KUKA KRL program: PPR-bot-01.src

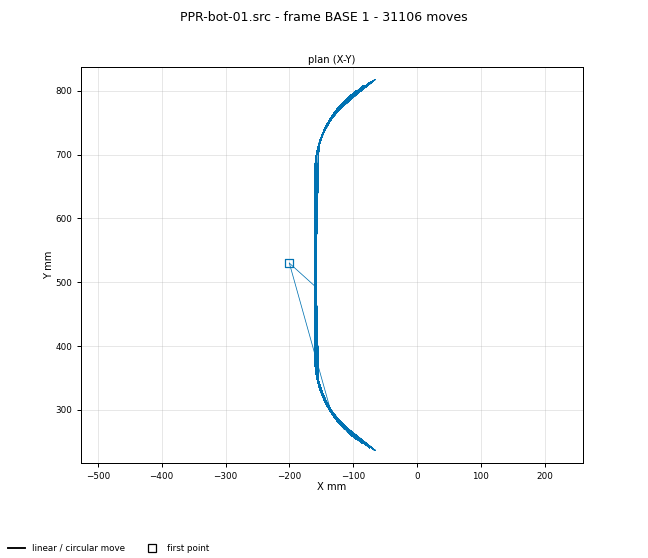
[picture p0: tool path of PPR-bot-01.src in frame BASE 1, 31106 of 31107 moves have a stored position in this frame; points joined in program order, loops and branches not executed]
&ACCESS RVEO
&REL 11
&PARAM TEMPLATE = C:\KRC\Roboter\Template\vorgabe
&PARAM EDITMASK = *
DEF variable_helical2( )
;FOLD INI
  ;FOLD BASISTECH INI
    GLOBAL INTERRUPT DECL 3 WHEN $STOPMESS==TRUE DO IR_STOPM ( )
    INTERRUPT ON 3
    BAS (#INITMOV,0 )
  ;ENDFOLD (BASISTECH INI)
 ;FOLD USER INI


    ;Make your modifications here
  ;ENDFOLD (USER INI)
;ENDFOLD (INI)
ACTION(#AXIS_RESET,34,1000,#NOERROR,ERROR_CODE)
;FOLD PTP HOME  Vel= 100 % DEFAULT;%{PE}%MKUKATPBASIS,%CMOVE,%VPTP,%P 1:PTP, 2:HOME, 3:, 5:100, 7:DEFAULT
$BWDSTART = FALSE
PDAT_ACT=PDEFAULT
FDAT_ACT=FHOME
BAS (#PTP_PARAMS,100 )
$H_POS=XHOME
PTP  XHOME
;ENDFOLD
BAS(#TOOL,1)
BAS(#BASE,1)
$VEL_AXIS[1]=100
$VEL_AXIS[2]=100
$VEL_AXIS[3]=100
$VEL_AXIS[4]=100
$VEL_AXIS[5]=100
$VEL_AXIS[6]=100
$VEL_EXTAX[1]=100
$VEL_EXTAX[2]=100

$ACC_AXIS[1]=100
$ACC_AXIS[2]=100
$ACC_AXIS[3]=100
$ACC_AXIS[4]=100
$ACC_AXIS[5]=100
$ACC_AXIS[6]=100
$ACC_EXTAX[1]=100
$ACC_EXTAX[2]=100

;;;;;;;;; postprocessing parameters (date 2024-01-25T18:13:03.555540)
; qxconst: -159.99
; qxconstarcys: -147.5,141.5
; qE3offset: 0.00
; qyoffset: 530.00
; qswitchsplit: 3
; qthinningtol: 0.2010
;;;;;;;;;

SLIN {X  -200.000, Y  +530.000, Z    +0.000, A    +0.000, E1    +0.000, E3    +0.000, E4    +0.000}

SLIN {X  -134.349, Y  +295.626, Z    +0.000, E1   +74.322, E3  -296.855}
HALT
SPLINE
SPL {X  -131.287, Y  +291.064, Z    +0.000, E1   +73.972, E3  -292.043}
SPL {X  -128.265, Y  +286.871, Z    +0.000, E1   +73.613, E3  -287.587}
SPL {X  -125.161, Y  +282.843, Z    +0.000, E1   +73.232, E3  -283.315}
SPL {X  -122.038, Y  +279.042, Z    +0.000, E1   +72.832, E3  -279.335}
SPL {X  -118.642, Y  +275.165, Z    +0.000, E1   +72.381, E3  -275.372}
SPL {X   -66.040, Y  +236.776, Z    +0.000, E1   +55.694, E3  -114.008}
ENDSPLINE

SPLINE
SPL {X  -127.452, Y  +285.790, Z    +0.000, E1   +56.591, E3   +59.937}
SPL {X  -151.591, Y  +331.344, Z    +0.000, E1   +43.870, E3   +76.036}
SPL {X  -158.135, Y  +358.205, Z    +0.000, E1   +26.984, E3   +79.764}
SPL {X  -159.602, Y  +371.361, Z    +0.000, E1   +14.835, E3   +80.660}
SPL {X  -159.981, Y  +380.818, Z    +0.000, E1    +4.512, E3   +80.938}
SPL {X  -159.990, Y  +384.681, Z    +0.000, E1    -0.222, E3   +80.967}
SPL {X  -159.990, Y  +387.626, Z    +0.000, E1    -8.190, E3   +80.995}
SPL {X  -159.990, Y  +390.340, Z    +0.000, E1   -15.987, E3   +81.060}
SPL {X  -159.990, Y  +394.216, Z    +0.000, E1   -27.062, E3   +81.222}
SPL {X  -159.990, Y  +399.855, Z    +0.000, E1   -40.916, E3   +81.593}
SPL {X  -159.990, Y  +405.475, Z    +0.000, E1   -51.039, E3   +82.110}
SPL {X  -159.990, Y  +414.231, Z    +0.000, E1   -60.575, E3   +83.294}
SPL {X  -159.990, Y  +462.953, Z    +0.000, E1   -73.611, E3   +95.033}
SPL {X  -153.839, Y  +715.436, Z    +0.000, E1   -75.884, E3  +197.463}
SPL {X  -148.840, Y  +730.182, Z    +0.000, E1   -75.434, E3  +210.040}
SPL {X  -143.409, Y  +742.426, Z    +0.000, E1   -74.905, E3  +221.552}
SPL {X  -139.557, Y  +749.735, Z    +0.000, E1   -74.483, E3  +228.900}
SPL {X  -136.371, Y  +755.165, Z    +0.000, E1   -74.152, E3  +234.446}
SPL {X  -133.102, Y  +760.274, Z    +0.000, E1   -73.777, E3  +239.831}
SPL {X  -128.975, Y  +766.169, Z    +0.000, E1   -73.313, E3  +246.106}
SPL {X  -124.947, Y  +771.425, Z    +0.000, E1   -72.782, E3  +251.799}
SPL {X  -121.698, Y  +775.357, Z    +0.000, E1   -72.353, E3  +255.994}
SPL {X  -118.622, Y  +778.858, Z    +0.000, E1   -71.924, E3  +259.620}
SPL {X   -66.171, Y  +817.165, Z    +0.000, E1   -56.016, E3  +410.978}
ENDSPLINE

SPLINE
SPL {X  -126.418, Y  +769.557, Z    +0.000, E1   -57.118, E3  +594.219}
SPL {X  -145.244, Y  +738.589, Z    +0.000, E1   -50.405, E3  +607.461}
SPL {X  -150.151, Y  +726.741, Z    +0.000, E1   -46.068, E3  +610.388}
SPL {X  -156.642, Y  +704.059, Z    +0.000, E1   -33.659, E3  +614.017}
SPL {X  -159.317, Y  +686.157, Z    +0.000, E1   -18.660, E3  +615.507}
SPL {X  -159.907, Y  +676.666, Z    +0.000, E1    -8.555, E3  +615.905}
SPL {X  -159.990, Y  +669.586, Z    +0.000, E1    -0.216, E3  +615.996}
SPL {X  -159.990, Y  +667.794, Z    +0.000, E1    +4.255, E3  +616.007}
SPL {X  -159.990, Y  +664.091, Z    +0.000, E1   +14.928, E3  +616.079}
SPL {X  -159.990, Y  +658.301, Z    +0.000, E1   +31.283, E3  +616.332}
SPL {X  -159.990, Y  +650.845, Z    +0.000, E1   +47.892, E3  +616.877}
SPL {X  -159.990, Y  +640.730, Z    +0.000, E1   +60.297, E3  +618.078}
SPL {X  -159.990, Y  +620.478, Z    +0.000, E1   +70.026, E3  +621.891}
SPL {X  -159.990, Y  +573.021, Z    +0.000, E1   +74.619, E3  +635.835}
SPL {X  -155.476, Y  +344.766, Z    +0.000, E1   +76.025, E3  +727.806}
SPL {X  -153.405, Y  +337.073, Z    +0.000, E1   +75.847, E3  +733.861}
SPL {X  -150.223, Y  +327.456, Z    +0.000, E1   +75.573, E3  +741.947}
SPL {X  -136.549, Y  +299.126, Z    +0.000, E1   +77.537, E3  +734.837}
ENDSPLINE

SPLINE
SPL {X  -136.626, Y  +299.252, Z    +0.000, E1   +76.314, E3  +746.487}
ENDSPLINE

SPLINE
SPL {X  -135.890, Y  +298.057, Z    +0.000, E1   +75.040, E3  +757.836}
SPL {X  -134.349, Y  +295.626, Z    +0.000, E1   +74.322, E3  +764.683}
SPL {X  -131.287, Y  +291.064, Z    +0.000, E1   +73.972, E3  +769.496}
SPL {X  -128.265, Y  +286.871, Z    +0.000, E1   +73.613, E3  +773.952}
SPL {X  -125.161, Y  +282.843, Z    +0.000, E1   +73.232, E3  +778.224}
SPL {X  -122.038, Y  +279.042, Z    +0.000, E1   +72.832, E3  +782.204}
SPL {X  -118.642, Y  +275.165, Z    +0.000, E1   +72.381, E3  +786.167}
SPL {X   -66.040, Y  +236.776, Z    +0.000, E1   +55.694, E3  +947.530}
ENDSPLINE

SPLINE
SPL {X  -127.452, Y  +285.790, Z    +0.000, E1   +56.591, E3 +1121.476}
SPL {X  -148.001, Y  +321.733, Z    +0.000, E1   +47.810, E3 +1135.579}
SPL {X  -154.604, Y  +341.337, Z    +0.000, E1   +38.630, E3 +1139.353}
SPL {X  -158.135, Y  +358.205, Z    +0.000, E1   +26.984, E3 +1141.302}
SPL {X  -159.602, Y  +371.361, Z    +0.000, E1   +14.835, E3 +1142.198}
SPL {X  -159.981, Y  +380.818, Z    +0.000, E1    +4.512, E3 +1142.476}
SPL {X  -159.990, Y  +384.681, Z    +0.000, E1    -0.222, E3 +1142.505}
SPL {X  -159.990, Y  +387.626, Z    +0.000, E1    -8.190, E3 +1142.534}
SPL {X  -159.990, Y  +390.340, Z    +0.000, E1   -15.987, E3 +1142.598}
SPL {X  -159.990, Y  +394.216, Z    +0.000, E1   -27.062, E3 +1142.760}
SPL {X  -159.990, Y  +399.855, Z    +0.000, E1   -40.916, E3 +1143.131}
SPL {X  -159.990, Y  +405.475, Z    +0.000, E1   -51.039, E3 +1143.648}
SPL {X  -159.990, Y  +414.231, Z    +0.000, E1   -60.575, E3 +1144.832}
SPL {X  -159.990, Y  +462.953, Z    +0.000, E1   -73.611, E3 +1156.571}
SPL {X  -153.839, Y  +715.436, Z    +0.000, E1   -75.884, E3 +1259.002}
SPL {X  -149.923, Y  +727.355, Z    +0.000, E1   -75.515, E3 +1269.112}
SPL {X  -145.995, Y  +736.939, Z    +0.000, E1   -75.150, E3 +1277.846}
SPL {X  -141.012, Y  +747.080, Z    +0.000, E1   -74.661, E3 +1287.699}
SPL {X  -136.371, Y  +755.165, Z    +0.000, E1   -74.152, E3 +1295.984}
SPL {X  -133.102, Y  +760.274, Z    +0.000, E1   -73.777, E3 +1301.369}
SPL {X  -128.975, Y  +766.169, Z    +0.000, E1   -73.313, E3 +1307.645}
SPL {X  -124.947, Y  +771.425, Z    +0.000, E1   -72.782, E3 +1313.338}
SPL {X  -121.698, Y  +775.357, Z    +0.000, E1   -72.353, E3 +1317.532}
SPL {X  -118.622, Y  +778.858, Z    +0.000, E1   -71.924, E3 +1321.158}
SPL {X   -66.171, Y  +817.165, Z    +0.000, E1   -56.016, E3 +1472.517}
ENDSPLINE

SPLINE
SPL {X  -126.418, Y  +769.557, Z    +0.000, E1   -57.118, E3 +1655.758}
SPL {X  -145.244, Y  +738.589, Z    +0.000, E1   -50.405, E3 +1668.999}
SPL {X  -150.151, Y  +726.741, Z    +0.000, E1   -46.068, E3 +1671.926}
SPL {X  -156.642, Y  +704.059, Z    +0.000, E1   -33.659, E3 +1675.555}
SPL {X  -159.317, Y  +686.157, Z    +0.000, E1   -18.660, E3 +1677.046}
SPL {X  -159.973, Y  +673.799, Z    +0.000, E1    -5.345, E3 +1677.494}
SPL {X  -159.990, Y  +669.500, Z    +0.000, E1    +0.000, E3 +1677.534}
SPL {X  -159.990, Y  +667.794, Z    +0.000, E1    +4.255, E3 +1677.546}
SPL {X  -159.990, Y  +664.091, Z    +0.000, E1   +14.928, E3 +1677.618}
SPL {X  -159.990, Y  +658.301, Z    +0.000, E1   +31.283, E3 +1677.870}
SPL {X  -159.990, Y  +650.845, Z    +0.000, E1   +47.892, E3 +1678.415}
SPL {X  -159.990, Y  +640.730, Z    +0.000, E1   +60.297, E3 +1679.617}
SPL {X  -159.990, Y  +620.478, Z    +0.000, E1   +70.026, E3 +1683.430}
SPL {X  -159.990, Y  +573.021, Z    +0.000, E1   +74.619, E3 +1697.374}
SPL {X  -154.165, Y  +339.724, Z    +0.000, E1   +75.927, E3 +1793.221}
SPL {X  -150.223, Y  +327.456, Z    +0.000, E1   +75.573, E3 +1803.486}
SPL {X  -136.549, Y  +299.126, Z    +0.000, E1   +77.537, E3 +1796.376}
ENDSPLINE

SPLINE
SPL {X  -136.862, Y  +299.641, Z    +0.000, E1   +76.604, E3 +1805.018}
ENDSPLINE

SPLINE
SPL {X  -136.434, Y  +298.938, Z    +0.000, E1   +75.982, E3 +1810.909}
SPL {X  -135.890, Y  +298.057, Z    +0.000, E1   +75.040, E3 +1819.375}
SPL {X  -134.349, Y  +295.626, Z    +0.000, E1   +74.322, E3 +1826.222}
SPL {X  -131.287, Y  +291.064, Z    +0.000, E1   +73.972, E3 +1831.034}
SPL {X  -128.265, Y  +286.871, Z    +0.000, E1   +73.613, E3 +1835.490}
SPL {X  -125.161, Y  +282.843, Z    +0.000, E1   +73.232, E3 +1839.762}
SPL {X  -122.038, Y  +279.042, Z    +0.000, E1   +72.832, E3 +1843.742}
SPL {X  -118.642, Y  +275.165, Z    +0.000, E1   +72.381, E3 +1847.705}
SPL {X   -66.040, Y  +236.776, Z    +0.000, E1   +55.694, E3 +2009.069}
ENDSPLINE

SPLINE
SPL {X  -127.452, Y  +285.790, Z    +0.000, E1   +56.591, E3 +2183.014}
SPL {X  -148.001, Y  +321.733, Z    +0.000, E1   +47.810, E3 +2197.118}
SPL {X  -154.604, Y  +341.337, Z    +0.000, E1   +38.630, E3 +2200.891}
SPL {X  -158.135, Y  +358.205, Z    +0.000, E1   +26.984, E3 +2202.841}
SPL {X  -159.602, Y  +371.361, Z    +0.000, E1   +14.835, E3 +2203.737}
SPL {X  -159.981, Y  +380.818, Z    +0.000, E1    +4.512, E3 +2204.015}
SPL {X  -159.990, Y  +384.681, Z    +0.000, E1    -0.222, E3 +2204.044}
SPL {X  -159.990, Y  +389.079, Z    +0.000, E1   -12.017, E3 +2204.107}
SPL {X  -159.990, Y  +394.216, Z    +0.000, E1   -27.062, E3 +2204.299}
SPL {X  -159.990, Y  +399.855, Z    +0.000, E1   -40.916, E3 +2204.670}
SPL {X  -159.990, Y  +405.475, Z    +0.000, E1   -51.039, E3 +2205.187}
SPL {X  -159.990, Y  +414.231, Z    +0.000, E1   -60.575, E3 +2206.371}
SPL {X  -159.990, Y  +462.953, Z    +0.000, E1   -73.611, E3 +2218.110}
SPL {X  -153.839, Y  +715.436, Z    +0.000, E1   -75.884, E3 +2320.540}
SPL {X  -148.840, Y  +730.182, Z    +0.000, E1   -75.434, E3 +2333.117}
SPL {X  -143.409, Y  +742.426, Z    +0.000, E1   -74.905, E3 +2344.629}
SPL {X  -139.557, Y  +749.735, Z    +0.000, E1   -74.483, E3 +2351.977}
SPL {X  -136.371, Y  +755.165, Z    +0.000, E1   -74.152, E3 +2357.523}
SPL {X  -133.102, Y  +760.274, Z    +0.000, E1   -73.777, E3 +2362.908}
SPL {X  -128.975, Y  +766.169, Z    +0.000, E1   -73.313, E3 +2369.183}
SPL {X  -124.947, Y  +771.425, Z    +0.000, E1   -72.782, E3 +2374.876}
SPL {X  -121.698, Y  +775.357, Z    +0.000, E1   -72.353, E3 +2379.071}
SPL {X  -118.622, Y  +778.858, Z    +0.000, E1   -71.924, E3 +2382.697}
SPL {X   -66.171, Y  +817.165, Z    +0.000, E1   -56.016, E3 +2534.055}
ENDSPLINE

SPLINE
SPL {X  -126.418, Y  +769.557, Z    +0.000, E1   -57.118, E3 +2717.296}
SPL {X  -145.244, Y  +738.589, Z    +0.000, E1   -50.405, E3 +2730.538}
SPL {X  -150.151, Y  +726.741, Z    +0.000, E1   -46.068, E3 +2733.464}
SPL {X  -156.642, Y  +704.059, Z    +0.000, E1   -33.659, E3 +2737.094}
SPL {X  -159.317, Y  +686.157, Z    +0.000, E1   -18.660, E3 +2738.584}
SPL {X  -159.973, Y  +673.799, Z    +0.000, E1    -5.345, E3 +2739.033}
SPL {X  -159.990, Y  +669.500, Z    +0.000, E1    +0.000, E3 +2739.073}
SPL {X  -159.990, Y  +667.794, Z    +0.000, E1    +4.255, E3 +2739.084}
SPL {X  -159.990, Y  +664.091, Z    +0.000, E1   +14.928, E3 +2739.156}
SPL {X  -159.990, Y  +658.301, Z    +0.000, E1   +31.283, E3 +2739.409}
SPL {X  -159.990, Y  +650.845, Z    +0.000, E1   +47.892, E3 +2739.954}
SPL {X  -159.990, Y  +640.730, Z    +0.000, E1   +60.297, E3 +2741.155}
SPL {X  -159.990, Y  +620.478, Z    +0.000, E1   +70.026, E3 +2744.968}
SPL {X  -159.990, Y  +573.021, Z    +0.000, E1   +74.619, E3 +2758.912}
SPL {X  -154.165, Y  +339.724, Z    +0.000, E1   +75.927, E3 +2854.759}
SPL {X  -150.223, Y  +327.456, Z    +0.000, E1   +75.573, E3 +2865.024}
SPL {X  -136.549, Y  +299.126, Z    +0.000, E1   +77.537, E3 +2857.914}
ENDSPLINE

SPLINE
SPL {X  -136.862, Y  +299.641, Z    +0.000, E1   +76.604, E3 +2866.556}
ENDSPLINE

SPLINE
SPL {X  -136.434, Y  +298.938, Z    +0.000, E1   +75.982, E3 +2872.447}
SPL {X  -135.890, Y  +298.057, Z    +0.000, E1   +75.040, E3 +2880.913}
SPL {X  -134.349, Y  +295.626, Z    +0.000, E1   +74.322, E3 +2887.760}
SPL {X  -131.287, Y  +291.064, Z    +0.000, E1   +73.972, E3 +2892.573}
SPL {X  -128.265, Y  +286.871, Z    +0.000, E1   +73.613, E3 +2897.029}
SPL {X  -125.161, Y  +282.843, Z    +0.000, E1   +73.232, E3 +2901.301}
SPL {X  -122.038, Y  +279.042, Z    +0.000, E1   +72.832, E3 +2905.281}
SPL {X  -118.642, Y  +275.165, Z    +0.000, E1   +72.381, E3 +2909.244}
SPL {X   -66.040, Y  +236.776, Z    +0.000, E1   +55.694, E3 +3070.607}
ENDSPLINE

SPLINE
SPL {X  -127.452, Y  +285.790, Z    +0.000, E1   +56.591, E3 +3244.552}
SPL {X  -148.001, Y  +321.733, Z    +0.000, E1   +47.810, E3 +3258.656}
SPL {X  -154.604, Y  +341.337, Z    +0.000, E1   +38.630, E3 +3262.430}
SPL {X  -158.135, Y  +358.205, Z    +0.000, E1   +26.984, E3 +3264.379}
SPL {X  -159.602, Y  +371.361, Z    +0.000, E1   +14.835, E3 +3265.275}
SPL {X  -159.981, Y  +380.818, Z    +0.000, E1    +4.512, E3 +3265.553}
SPL {X  -159.990, Y  +384.681, Z    +0.000, E1    -0.222, E3 +3265.582}
SPL {X  -159.990, Y  +389.079, Z    +0.000, E1   -12.017, E3 +3265.645}
SPL {X  -159.990, Y  +394.216, Z    +0.000, E1   -27.062, E3 +3265.837}
SPL {X  -159.990, Y  +399.855, Z    +0.000, E1   -40.916, E3 +3266.208}
SPL {X  -159.990, Y  +405.475, Z    +0.000, E1   -51.039, E3 +3266.725}
SPL {X  -159.990, Y  +414.231, Z    +0.000, E1   -60.575, E3 +3267.909}
SPL {X  -159.990, Y  +462.953, Z    +0.000, E1   -73.611, E3 +3279.648}
SPL {X  -153.839, Y  +715.436, Z    +0.000, E1   -75.884, E3 +3382.079}
SPL {X  -148.840, Y  +730.182, Z    +0.000, E1   -75.434, E3 +3394.655}
SPL {X  -143.409, Y  +742.426, Z    +0.000, E1   -74.905, E3 +3406.167}
SPL {X  -139.557, Y  +749.735, Z    +0.000, E1   -74.483, E3 +3413.515}
SPL {X  -136.371, Y  +755.165, Z    +0.000, E1   -74.152, E3 +3419.061}
SPL {X  -133.102, Y  +760.274, Z    +0.000, E1   -73.777, E3 +3424.446}
SPL {X  -128.975, Y  +766.169, Z    +0.000, E1   -73.313, E3 +3430.722}
SPL {X  -124.947, Y  +771.425, Z    +0.000, E1   -72.782, E3 +3436.415}
SPL {X  -121.698, Y  +775.357, Z    +0.000, E1   -72.353, E3 +3440.609}
SPL {X  -118.622, Y  +778.858, Z    +0.000, E1   -71.924, E3 +3444.235}
SPL {X   -66.171, Y  +817.165, Z    +0.000, E1   -56.016, E3 +3595.593}
ENDSPLINE

SPLINE
SPL {X  -126.418, Y  +769.557, Z    +0.000, E1   -57.118, E3 +3778.835}
SPL {X  -145.244, Y  +738.589, Z    +0.000, E1   -50.405, E3 +3792.076}
SPL {X  -150.151, Y  +726.741, Z    +0.000, E1   -46.068, E3 +3795.003}
SPL {X  -156.642, Y  +704.059, Z    +0.000, E1   -33.659, E3 +3798.632}
SPL {X  -159.317, Y  +686.157, Z    +0.000, E1   -18.660, E3 +3800.123}
SPL {X  -159.973, Y  +673.799, Z    +0.000, E1    -5.345, E3 +3800.571}
SPL {X  -159.990, Y  +669.500, Z    +0.000, E1    +0.000, E3 +3800.611}
SPL {X  -159.990, Y  +667.794, Z    +0.000, E1    +4.255, E3 +3800.623}
SPL {X  -159.990, Y  +664.091, Z    +0.000, E1   +14.928, E3 +3800.695}
SPL {X  -159.990, Y  +658.301, Z    +0.000, E1   +31.283, E3 +3800.947}
SPL {X  -159.990, Y  +650.845, Z    +0.000, E1   +47.892, E3 +3801.492}
SPL {X  -159.990, Y  +640.730, Z    +0.000, E1   +60.297, E3 +3802.693}
SPL {X  -159.990, Y  +620.478, Z    +0.000, E1   +70.026, E3 +3806.507}
SPL {X  -159.990, Y  +573.021, Z    +0.000, E1   +74.619, E3 +3820.451}
SPL {X  -154.165, Y  +339.724, Z    +0.000, E1   +75.927, E3 +3916.298}
SPL {X  -150.223, Y  +327.456, Z    +0.000, E1   +75.573, E3 +3926.562}
SPL {X  -136.549, Y  +299.126, Z    +0.000, E1   +77.537, E3 +3919.452}
ENDSPLINE

SPLINE
SPL {X  -136.862, Y  +299.641, Z    +0.000, E1   +76.604, E3 +3928.094}
ENDSPLINE

SPLINE
SPL {X  -136.434, Y  +298.938, Z    +0.000, E1   +75.982, E3 +3933.986}
SPL {X  -135.890, Y  +298.057, Z    +0.000, E1   +75.040, E3 +3942.452}
SPL {X  -134.349, Y  +295.626, Z    +0.000, E1   +74.322, E3 +3949.299}
SPL {X  -131.287, Y  +291.064, Z    +0.000, E1   +73.972, E3 +3954.111}
SPL {X  -128.265, Y  +286.871, Z    +0.000, E1   +73.613, E3 +3958.567}
SPL {X  -125.161, Y  +282.843, Z    +0.000, E1   +73.232, E3 +3962.839}
SPL {X  -122.038, Y  +279.042, Z    +0.000, E1   +72.832, E3 +3966.819}
SPL {X  -118.642, Y  +275.165, Z    +0.000, E1   +72.381, E3 +3970.782}
SPL {X   -66.040, Y  +236.776, Z    +0.000, E1   +55.694, E3 +4132.146}
ENDSPLINE

SPLINE
SPL {X  -127.452, Y  +285.790, Z    +0.000, E1   +56.591, E3 +4306.091}
SPL {X  -148.001, Y  +321.733, Z    +0.000, E1   +47.810, E3 +4320.194}
SPL {X  -154.604, Y  +341.337, Z    +0.000, E1   +38.630, E3 +4323.968}
SPL {X  -158.135, Y  +358.205, Z    +0.000, E1   +26.984, E3 +4325.918}
SPL {X  -159.602, Y  +371.361, Z    +0.000, E1   +14.835, E3 +4326.814}
SPL {X  -159.981, Y  +380.818, Z    +0.000, E1    +4.512, E3 +4327.092}
SPL {X  -159.990, Y  +384.681, Z    +0.000, E1    -0.222, E3 +4327.121}
SPL {X  -159.990, Y  +389.079, Z    +0.000, E1   -12.017, E3 +4327.184}
SPL {X  -159.990, Y  +394.216, Z    +0.000, E1   -27.062, E3 +4327.375}
SPL {X  -159.990, Y  +399.855, Z    +0.000, E1   -40.916, E3 +4327.747}
SPL {X  -159.990, Y  +405.475, Z    +0.000, E1   -51.039, E3 +4328.263}
SPL {X  -159.990, Y  +414.231, Z    +0.000, E1   -60.575, E3 +4329.448}
SPL {X  -159.990, Y  +462.953, Z    +0.000, E1   -73.611, E3 +4341.187}
SPL {X  -153.839, Y  +715.436, Z    +0.000, E1   -75.884, E3 +4443.617}
SPL {X  -148.840, Y  +730.182, Z    +0.000, E1   -75.434, E3 +4456.194}
SPL {X  -143.409, Y  +742.426, Z    +0.000, E1   -74.905, E3 +4467.706}
SPL {X  -139.557, Y  +749.735, Z    +0.000, E1   -74.483, E3 +4475.054}
SPL {X  -136.371, Y  +755.165, Z    +0.000, E1   -74.152, E3 +4480.600}
SPL {X  -133.102, Y  +760.274, Z    +0.000, E1   -73.777, E3 +4485.985}
SPL {X  -128.975, Y  +766.169, Z    +0.000, E1   -73.313, E3 +4492.260}
SPL {X  -124.947, Y  +771.425, Z    +0.000, E1   -72.782, E3 +4497.953}
SPL {X  -121.698, Y  +775.357, Z    +0.000, E1   -72.353, E3 +4502.148}
SPL {X  -118.622, Y  +778.858, Z    +0.000, E1   -71.924, E3 +4505.774}
SPL {X   -66.171, Y  +817.165, Z    +0.000, E1   -56.016, E3 +4657.132}
ENDSPLINE

SPLINE
SPL {X  -126.418, Y  +769.557, Z    +0.000, E1   -57.118, E3 +4840.373}
SPL {X  -145.244, Y  +738.589, Z    +0.000, E1   -50.405, E3 +4853.615}
SPL {X  -150.151, Y  +726.741, Z    +0.000, E1   -46.068, E3 +4856.541}
SPL {X  -156.642, Y  +704.059, Z    +0.000, E1   -33.659, E3 +4860.171}
SPL {X  -159.317, Y  +686.157, Z    +0.000, E1   -18.660, E3 +4861.661}
SPL {X  -159.973, Y  +673.799, Z    +0.000, E1    -5.345, E3 +4862.110}
SPL {X  -159.990, Y  +669.500, Z    +0.000, E1    +0.000, E3 +4862.150}
SPL {X  -159.990, Y  +667.794, Z    +0.000, E1    +4.255, E3 +4862.161}
SPL {X  -159.990, Y  +664.091, Z    +0.000, E1   +14.928, E3 +4862.233}
SPL {X  -159.990, Y  +658.301, Z    +0.000, E1   +31.283, E3 +4862.486}
SPL {X  -159.990, Y  +650.845, Z    +0.000, E1   +47.892, E3 +4863.031}
SPL {X  -159.990, Y  +640.730, Z    +0.000, E1   +60.297, E3 +4864.232}
SPL {X  -159.990, Y  +620.478, Z    +0.000, E1   +70.026, E3 +4868.045}
SPL {X  -159.990, Y  +573.021, Z    +0.000, E1   +74.619, E3 +4881.989}
SPL {X  -154.165, Y  +339.724, Z    +0.000, E1   +75.927, E3 +4977.836}
SPL {X  -150.223, Y  +327.456, Z    +0.000, E1   +75.573, E3 +4988.101}
SPL {X  -136.549, Y  +299.126, Z    +0.000, E1   +77.537, E3 +4980.991}
ENDSPLINE

SPLINE
SPL {X  -136.862, Y  +299.641, Z    +0.000, E1   +76.604, E3 +4989.633}
ENDSPLINE

SPLINE
SPL {X  -136.434, Y  +298.938, Z    +0.000, E1   +75.982, E3 +4995.524}
SPL {X  -135.890, Y  +298.057, Z    +0.000, E1   +75.040, E3 +5003.990}
SPL {X  -134.349, Y  +295.626, Z    +0.000, E1   +74.322, E3 +5010.837}
SPL {X  -131.287, Y  +291.064, Z    +0.000, E1   +73.972, E3 +5015.650}
SPL {X  -128.265, Y  +286.871, Z    +0.000, E1   +73.613, E3 +5020.106}
SPL {X  -125.161, Y  +282.843, Z    +0.000, E1   +73.232, E3 +5024.378}
SPL {X  -122.038, Y  +279.042, Z    +0.000, E1   +72.832, E3 +5028.357}
SPL {X  -118.642, Y  +275.165, Z    +0.000, E1   +72.381, E3 +5032.321}
SPL {X   -66.040, Y  +236.776, Z    +0.000, E1   +55.694, E3 +5193.684}
ENDSPLINE

SPLINE
SPL {X  -127.452, Y  +285.790, Z    +0.000, E1   +56.591, E3 +5367.629}
SPL {X  -151.591, Y  +331.344, Z    +0.000, E1   +43.870, E3 +5383.729}
SPL {X  -158.135, Y  +358.205, Z    +0.000, E1   +26.984, E3 +5387.456}
SPL {X  -159.602, Y  +371.361, Z    +0.000, E1   +14.835, E3 +5388.352}
SPL {X  -159.981, Y  +380.818, Z    +0.000, E1    +4.512, E3 +5388.630}
SPL {X  -159.990, Y  +384.681, Z    +0.000, E1    -0.222, E3 +5388.659}
SPL {X  -159.990, Y  +387.626, Z    +0.000, E1    -8.190, E3 +5388.687}
SPL {X  -159.990, Y  +390.340, Z    +0.000, E1   -15.987, E3 +5388.752}
SPL {X  -159.990, Y  +394.216, Z    +0.000, E1   -27.062, E3 +5388.914}
SPL {X  -159.990, Y  +399.855, Z    +0.000, E1   -40.916, E3 +5389.285}
SPL {X  -159.990, Y  +405.475, Z    +0.000, E1   -51.039, E3 +5389.802}
SPL {X  -159.990, Y  +414.231, Z    +0.000, E1   -60.575, E3 +5390.986}
SPL {X  -159.990, Y  +462.953, Z    +0.000, E1   -73.611, E3 +5402.725}
SPL {X  -153.839, Y  +715.436, Z    +0.000, E1   -75.884, E3 +5505.156}
SPL {X  -149.923, Y  +727.355, Z    +0.000, E1   -75.515, E3 +5515.266}
SPL {X  -145.995, Y  +736.939, Z    +0.000, E1   -75.150, E3 +5524.000}
SPL {X  -141.012, Y  +747.080, Z    +0.000, E1   -74.661, E3 +5533.853}
SPL {X  -136.371, Y  +755.165, Z    +0.000, E1   -74.152, E3 +5542.138}
SPL {X  -131.455, Y  +762.694, Z    +0.000, E1   -73.615, E3 +5550.056}
SPL {X  -125.933, Y  +770.180, Z    +0.000, E1   -72.934, E3 +5558.121}
SPL {X  -121.698, Y  +775.357, Z    +0.000, E1   -72.353, E3 +5563.686}
SPL {X  -118.622, Y  +778.858, Z    +0.000, E1   -71.924, E3 +5567.312}
SPL {X   -66.171, Y  +817.165, Z    +0.000, E1   -56.016, E3 +5718.670}
ENDSPLINE

SPLINE
SPL {X  -126.418, Y  +769.557, Z    +0.000, E1   -57.118, E3 +5901.912}
SPL {X  -145.244, Y  +738.589, Z    +0.000, E1   -50.405, E3 +5915.153}
SPL {X  -150.151, Y  +726.741, Z    +0.000, E1   -46.068, E3 +5918.080}
SPL {X  -156.642, Y  +704.059, Z    +0.000, E1   -33.659, E3 +5921.709}
SPL {X  -159.317, Y  +686.157, Z    +0.000, E1   -18.660, E3 +5923.200}
SPL {X  -159.973, Y  +673.799, Z    +0.000, E1    -5.345, E3 +5923.648}
SPL {X  -159.990, Y  +669.500, Z    +0.000, E1    +0.000, E3 +5923.688}
SPL {X  -159.990, Y  +667.794, Z    +0.000, E1    +4.255, E3 +5923.699}
SPL {X  -159.990, Y  +664.091, Z    +0.000, E1   +14.928, E3 +5923.772}
SPL {X  -159.990, Y  +658.301, Z    +0.000, E1   +31.283, E3 +5924.024}
SPL {X  -159.990, Y  +650.845, Z    +0.000, E1   +47.892, E3 +5924.569}
SPL {X  -159.990, Y  +640.730, Z    +0.000, E1   +60.297, E3 +5925.770}
SPL {X  -159.990, Y  +620.478, Z    +0.000, E1   +70.026, E3 +5929.584}
SPL {X  -159.990, Y  +573.021, Z    +0.000, E1   +74.619, E3 +5943.528}
SPL {X  -154.165, Y  +339.724, Z    +0.000, E1   +75.927, E3 +6039.374}
SPL {X  -150.223, Y  +327.456, Z    +0.000, E1   +75.573, E3 +6049.639}
SPL {X  -136.549, Y  +299.126, Z    +0.000, E1   +77.537, E3 +6042.529}
ENDSPLINE

SPLINE
SPL {X  -136.862, Y  +299.641, Z    +0.000, E1   +76.604, E3 +6051.171}
ENDSPLINE

SPLINE
SPL {X  -136.434, Y  +298.938, Z    +0.000, E1   +75.982, E3 +6057.062}
SPL {X  -135.890, Y  +298.057, Z    +0.000, E1   +75.040, E3 +6065.528}
SPL {X  -134.349, Y  +295.626, Z    +0.000, E1   +74.322, E3 +6072.376}
SPL {X  -131.287, Y  +291.064, Z    +0.000, E1   +73.972, E3 +6077.188}
SPL {X  -128.265, Y  +286.871, Z    +0.000, E1   +73.613, E3 +6081.644}
SPL {X  -125.161, Y  +282.843, Z    +0.000, E1   +73.232, E3 +6085.916}
SPL {X  -122.038, Y  +279.042, Z    +0.000, E1   +72.832, E3 +6089.896}
SPL {X  -118.642, Y  +275.165, Z    +0.000, E1   +72.381, E3 +6093.859}
SPL {X   -66.040, Y  +236.776, Z    +0.000, E1   +55.694, E3 +6255.223}
ENDSPLINE

SPLINE
SPL {X  -127.452, Y  +285.790, Z    +0.000, E1   +56.591, E3 +6429.168}
SPL {X  -151.591, Y  +331.344, Z    +0.000, E1   +43.870, E3 +6445.267}
SPL {X  -158.135, Y  +358.205, Z    +0.000, E1   +26.984, E3 +6448.995}
SPL {X  -159.602, Y  +371.361, Z    +0.000, E1   +14.835, E3 +6449.891}
SPL {X  -159.981, Y  +380.818, Z    +0.000, E1    +4.512, E3 +6450.169}
SPL {X  -159.990, Y  +384.681, Z    +0.000, E1    -0.222, E3 +6450.198}
SPL {X  -159.990, Y  +389.079, Z    +0.000, E1   -12.017, E3 +6450.261}
SPL {X  -159.990, Y  +394.216, Z    +0.000, E1   -27.062, E3 +6450.452}
SPL {X  -159.990, Y  +399.855, Z    +0.000, E1   -40.916, E3 +6450.823}
SPL {X  -159.990, Y  +405.475, Z    +0.000, E1   -51.039, E3 +6451.340}
SPL {X  -159.990, Y  +414.231, Z    +0.000, E1   -60.575, E3 +6452.525}
SPL {X  -159.990, Y  +462.953, Z    +0.000, E1   -73.611, E3 +6464.264}
SPL {X  -153.839, Y  +715.436, Z    +0.000, E1   -75.884, E3 +6566.694}
SPL {X  -148.840, Y  +730.182, Z    +0.000, E1   -75.434, E3 +6579.271}
SPL {X  -143.409, Y  +742.426, Z    +0.000, E1   -74.905, E3 +6590.783}
SPL {X  -139.557, Y  +749.735, Z    +0.000, E1   -74.483, E3 +6598.131}
SPL {X  -136.371, Y  +755.165, Z    +0.000, E1   -74.152, E3 +6603.677}
SPL {X  -131.455, Y  +762.694, Z    +0.000, E1   -73.615, E3 +6611.595}
SPL {X  -125.933, Y  +770.180, Z    +0.000, E1   -72.934, E3 +6619.659}
SPL {X  -121.698, Y  +775.357, Z    +0.000, E1   -72.353, E3 +6625.225}
SPL {X  -118.622, Y  +778.858, Z    +0.000, E1   -71.924, E3 +6628.851}
SPL {X   -66.171, Y  +817.165, Z    +0.000, E1   -56.016, E3 +6780.209}
ENDSPLINE

SPLINE
SPL {X  -126.418, Y  +769.557, Z    +0.000, E1   -57.118, E3 +6963.450}
SPL {X  -148.476, Y  +731.097, Z    +0.000, E1   -47.824, E3 +6978.606}
SPL {X  -156.642, Y  +704.059, Z    +0.000, E1   -33.659, E3 +6983.248}
SPL {X  -159.317, Y  +686.157, Z    +0.000, E1   -18.660, E3 +6984.738}
SPL {X  -159.907, Y  +676.666, Z    +0.000, E1    -8.555, E3 +6985.136}
SPL {X  -159.990, Y  +669.586, Z    +0.000, E1    -0.216, E3 +6985.226}
SPL {X  -159.990, Y  +667.794, Z    +0.000, E1    +4.255, E3 +6985.238}
SPL {X  -159.990, Y  +664.091, Z    +0.000, E1   +14.928, E3 +6985.310}
SPL {X  -159.990, Y  +659.599, Z    +0.000, E1   +28.016, E3 +6985.480}
SPL {X  -159.990, Y  +652.711, Z    +0.000, E1   +44.293, E3 +6985.960}
SPL {X  -159.990, Y  +640.730, Z    +0.000, E1   +60.297, E3 +6987.309}
SPL {X  -159.990, Y  +620.478, Z    +0.000, E1   +70.026, E3 +6991.122}
SPL {X  -159.990, Y  +573.021, Z    +0.000, E1   +74.619, E3 +7005.066}
SPL {X  -154.165, Y  +339.724, Z    +0.000, E1   +75.927, E3 +7100.913}
SPL {X  -150.223, Y  +327.456, Z    +0.000, E1   +75.573, E3 +7111.178}
SPL {X  -136.549, Y  +299.126, Z    +0.000, E1   +77.537, E3 +7104.068}
ENDSPLINE

SPLINE
SPL {X  -136.862, Y  +299.641, Z    +0.000, E1   +76.604, E3 +7112.710}
ENDSPLINE

SPLINE
SPL {X  -136.434, Y  +298.938, Z    +0.000, E1   +75.982, E3 +7118.601}
SPL {X  -135.890, Y  +298.057, Z    +0.000, E1   +75.040, E3 +7127.067}
SPL {X  -134.349, Y  +295.626, Z    +0.000, E1   +74.322, E3 +7133.914}
SPL {X  -131.287, Y  +291.064, Z    +0.000, E1   +73.972, E3 +7138.727}
SPL {X  -128.265, Y  +286.871, Z    +0.000, E1   +73.613, E3 +7143.183}
SPL {X  -125.161, Y  +282.843, Z    +0.000, E1   +73.232, E3 +7147.454}
SPL {X  -122.038, Y  +279.042, Z    +0.000, E1   +72.832, E3 +7151.434}
SPL {X  -118.642, Y  +275.165, Z    +0.000, E1   +72.381, E3 +7155.398}
SPL {X   -66.040, Y  +236.776, Z    +0.000, E1   +55.694, E3 +7316.761}
ENDSPLINE

SPLINE
SPL {X  -127.452, Y  +285.790, Z    +0.000, E1   +56.591, E3 +7490.706}
SPL {X  -151.591, Y  +331.344, Z    +0.000, E1   +43.870, E3 +7506.806}
SPL {X  -158.135, Y  +358.205, Z    +0.000, E1   +26.984, E3 +7510.533}
SPL {X  -159.602, Y  +371.361, Z    +0.000, E1   +14.835, E3 +7511.429}
SPL {X  -159.981, Y  +380.818, Z    +0.000, E1    +4.512, E3 +7511.707}
SPL {X  -159.990, Y  +384.681, Z    +0.000, E1    -0.222, E3 +7511.736}
SPL {X  -159.990, Y  +387.626, Z    +0.000, E1    -8.190, E3 +7511.764}
SPL {X  -159.990, Y  +390.340, Z    +0.000, E1   -15.987, E3 +7511.829}
SPL {X  -159.990, Y  +394.216, Z    +0.000, E1   -27.062, E3 +7511.991}
SPL {X  -159.990, Y  +399.855, Z    +0.000, E1   -40.916, E3 +7512.362}
SPL {X  -159.990, Y  +405.475, Z    +0.000, E1   -51.039, E3 +7512.879}
SPL {X  -159.990, Y  +414.231, Z    +0.000, E1   -60.575, E3 +7514.063}
SPL {X  -159.990, Y  +462.953, Z    +0.000, E1   -73.611, E3 +7525.802}
SPL {X  -153.839, Y  +715.436, Z    +0.000, E1   -75.884, E3 +7628.233}
SPL {X  -148.840, Y  +730.182, Z    +0.000, E1   -75.434, E3 +7640.809}
SPL {X  -143.409, Y  +742.426, Z    +0.000, E1   -74.905, E3 +7652.321}
SPL {X  -139.557, Y  +749.735, Z    +0.000, E1   -74.483, E3 +7659.669}
SPL {X  -136.371, Y  +755.165, Z    +0.000, E1   -74.152, E3 +7665.215}
SPL {X  -133.102, Y  +760.274, Z    +0.000, E1   -73.777, E3 +7670.600}
SPL {X  -128.975, Y  +766.169, Z    +0.000, E1   -73.313, E3 +7676.875}
SPL {X  -124.947, Y  +771.425, Z    +0.000, E1   -72.782, E3 +7682.568}
SPL {X  -121.698, Y  +775.357, Z    +0.000, E1   -72.353, E3 +7686.763}
SPL {X  -118.622, Y  +778.858, Z    +0.000, E1   -71.924, E3 +7690.389}
SPL {X   -66.171, Y  +817.165, Z    +0.000, E1   -56.016, E3 +7841.747}
ENDSPLINE

SPLINE
SPL {X  -126.418, Y  +769.557, Z    +0.000, E1   -57.118, E3 +8024.989}
SPL {X  -145.244, Y  +738.589, Z    +0.000, E1   -50.405, E3 +8038.230}
SPL {X  -150.151, Y  +726.741, Z    +0.000, E1   -46.068, E3 +8041.157}
SPL {X  -156.642, Y  +704.059, Z    +0.000, E1   -33.659, E3 +8044.786}
SPL {X  -159.317, Y  +686.157, Z    +0.000, E1   -18.660, E3 +8046.276}
SPL {X  -159.907, Y  +676.666, Z    +0.000, E1    -8.555, E3 +8046.674}
SPL {X  -159.990, Y  +669.586, Z    +0.000, E1    -0.216, E3 +8046.765}
SPL {X  -159.990, Y  +667.794, Z    +0.000, E1    +4.255, E3 +8046.776}
SPL {X  -159.990, Y  +664.091, Z    +0.000, E1   +14.928, E3 +8046.848}
SPL {X  -159.990, Y  +659.599, Z    +0.000, E1   +28.016, E3 +8047.019}
SPL {X  -159.990, Y  +652.711, Z    +0.000, E1   +44.293, E3 +8047.498}
SPL {X  -159.990, Y  +640.730, Z    +0.000, E1   +60.297, E3 +8048.847}
SPL {X  -159.990, Y  +620.478, Z    +0.000, E1   +70.026, E3 +8052.661}
SPL {X  -159.990, Y  +573.021, Z    +0.000, E1   +74.619, E3 +8066.604}
SPL {X  -154.165, Y  +339.724, Z    +0.000, E1   +75.927, E3 +8162.451}
SPL {X  -150.223, Y  +327.456, Z    +0.000, E1   +75.573, E3 +8172.716}
SPL {X  -136.549, Y  +299.126, Z    +0.000, E1   +77.537, E3 +8165.606}
ENDSPLINE

SPLINE
SPL {X  -136.626, Y  +299.252, Z    +0.000, E1   +76.314, E3 +8177.256}
ENDSPLINE

SPLINE
SPL {X  -135.890, Y  +298.057, Z    +0.000, E1   +75.040, E3 +8188.605}
SPL {X  -134.349, Y  +295.626, Z    +0.000, E1   +74.322, E3 +8195.453}
SPL {X  -131.287, Y  +291.064, Z    +0.000, E1   +73.972, E3 +8200.265}
SPL {X  -128.265, Y  +286.871, Z    +0.000, E1   +73.613, E3 +8204.721}
SPL {X  -125.161, Y  +282.843, Z    +0.000, E1   +73.232, E3 +8208.993}
SPL {X  -122.038, Y  +279.042, Z    +0.000, E1   +72.832, E3 +8212.973}
SPL {X  -118.642, Y  +275.165, Z    +0.000, E1   +72.381, E3 +8216.936}
SPL {X   -66.040, Y  +236.776, Z    +0.000, E1   +55.694, E3 +8378.299}
ENDSPLINE

SPLINE
SPL {X  -127.452, Y  +285.790, Z    +0.000, E1   +56.591, E3 +8552.245}
SPL {X  -151.591, Y  +331.344, Z    +0.000, E1   +43.870, E3 +8568.344}
SPL {X  -158.135, Y  +358.205, Z    +0.000, E1   +26.984, E3 +8572.072}
SPL {X  -159.602, Y  +371.361, Z    +0.000, E1   +14.835, E3 +8572.968}
SPL {X  -159.981, Y  +380.818, Z    +0.000, E1    +4.512, E3 +8573.246}
SPL {X  -159.990, Y  +384.681, Z    +0.000, E1    -0.222, E3 +8573.274}
SPL {X  -159.990, Y  +389.079, Z    +0.000, E1   -12.017, E3 +8573.337}
SPL {X  -159.990, Y  +394.216, Z    +0.000, E1   -27.062, E3 +8573.529}
SPL {X  -159.990, Y  +401.720, Z    +0.000, E1   -44.434, E3 +8574.072}
SPL {X  -159.990, Y  +414.231, Z    +0.000, E1   -60.575, E3 +8575.602}
SPL {X  -159.990, Y  +462.953, Z    +0.000, E1   -73.611, E3 +8587.341}
SPL {X  -153.839, Y  +715.436, Z    +0.000, E1   -75.884, E3 +8689.771}
SPL {X  -148.840, Y  +730.182, Z    +0.000, E1   -75.434, E3 +8702.348}
SPL {X  -143.409, Y  +742.426, Z    +0.000, E1   -74.905, E3 +8713.860}
SPL {X  -139.557, Y  +749.735, Z    +0.000, E1   -74.483, E3 +8721.208}
SPL {X  -136.371, Y  +755.165, Z    +0.000, E1   -74.152, E3 +8726.753}
SPL {X  -131.455, Y  +762.694, Z    +0.000, E1   -73.615, E3 +8734.672}
SPL {X  -125.933, Y  +770.180, Z    +0.000, E1   -72.934, E3 +8742.736}
SPL {X  -121.698, Y  +775.357, Z    +0.000, E1   -72.353, E3 +8748.301}
SPL {X  -118.622, Y  +778.858, Z    +0.000, E1   -71.924, E3 +8751.927}
SPL {X   -66.171, Y  +817.165, Z    +0.000, E1   -56.016, E3 +8903.286}
ENDSPLINE

SPLINE
SPL {X  -126.418, Y  +769.557, Z    +0.000, E1   -57.118, E3 +9086.527}
SPL {X  -145.244, Y  +738.589, Z    +0.000, E1   -50.405, E3 +9099.769}
SPL {X  -150.151, Y  +726.741, Z    +0.000, E1   -46.068, E3 +9102.695}
SPL {X  -156.642, Y  +704.059, Z    +0.000, E1   -33.659, E3 +9106.325}
SPL {X  -159.317, Y  +686.157, Z    +0.000, E1   -18.660, E3 +9107.815}
SPL {X  -159.973, Y  +673.799, Z    +0.000, E1    -5.345, E3 +9108.264}
SPL {X  -159.990, Y  +669.500, Z    +0.000, E1    +0.000, E3 +9108.304}
SPL {X  -159.990, Y  +667.794, Z    +0.000, E1    +4.255, E3 +9108.315}
SPL {X  -159.990, Y  +664.091, Z    +0.000, E1   +14.928, E3 +9108.387}
SPL {X  -159.990, Y  +659.599, Z    +0.000, E1   +28.016, E3 +9108.557}
SPL {X  -159.990, Y  +652.711, Z    +0.000, E1   +44.293, E3 +9109.037}
SPL {X  -159.990, Y  +640.730, Z    +0.000, E1   +60.297, E3 +9110.386}
SPL {X  -159.990, Y  +620.478, Z    +0.000, E1   +70.026, E3 +9114.199}
SPL {X  -159.990, Y  +573.021, Z    +0.000, E1   +74.619, E3 +9128.143}
SPL {X  -154.165, Y  +339.724, Z    +0.000, E1   +75.927, E3 +9223.990}
SPL {X  -150.571, Y  +328.416, Z    +0.000, E1   +75.599, E3 +9233.435}
SPL {X  -148.206, Y  +322.236, Z    +0.000, E1   +75.365, E3 +9238.979}
SPL {X  -136.549, Y  +299.126, Z    +0.000, E1   +77.537, E3 +9227.145}
ENDSPLINE

SPLINE
SPL {X  -136.862, Y  +299.641, Z    +0.000, E1   +76.604, E3 +9235.787}
ENDSPLINE

SPLINE
SPL {X  -136.434, Y  +298.938, Z    +0.000, E1   +75.982, E3 +9241.678}
SPL {X  -135.890, Y  +298.057, Z    +0.000, E1   +75.040, E3 +9250.144}
SPL {X  -134.349, Y  +295.626, Z    +0.000, E1   +74.322, E3 +9256.991}
SPL {X  -131.287, Y  +291.064, Z    +0.000, E1   +73.972, E3 +9261.804}
SPL {X  -128.265, Y  +286.871, Z    +0.000, E1   +73.613, E3 +9266.260}
SPL {X  -125.161, Y  +282.843, Z    +0.000, E1   +73.232, E3 +9270.531}
SPL {X  -122.038, Y  +279.042, Z    +0.000, E1   +72.832, E3 +9274.511}
SPL {X  -118.642, Y  +275.165, Z    +0.000, E1   +72.381, E3 +9278.474}
SPL {X   -66.040, Y  +236.776, Z    +0.000, E1   +55.694, E3 +9439.838}
ENDSPLINE

SPLINE
SPL {X  -127.452, Y  +285.790, Z    +0.000, E1   +56.591, E3 +9613.783}
SPL {X  -151.591, Y  +331.344, Z    +0.000, E1   +43.870, E3 +9629.883}
SPL {X  -158.135, Y  +358.205, Z    +0.000, E1   +26.984, E3 +9633.610}
SPL {X  -159.602, Y  +371.361, Z    +0.000, E1   +14.835, E3 +9634.506}
SPL {X  -159.981, Y  +380.818, Z    +0.000, E1    +4.512, E3 +9634.784}
SPL {X  -159.990, Y  +384.681, Z    +0.000, E1    -0.222, E3 +9634.813}
SPL {X  -159.990, Y  +387.626, Z    +0.000, E1    -8.190, E3 +9634.841}
SPL {X  -159.990, Y  +390.340, Z    +0.000, E1   -15.987, E3 +9634.906}
SPL {X  -159.990, Y  +394.216, Z    +0.000, E1   -27.062, E3 +9635.068}
SPL {X  -159.990, Y  +399.855, Z    +0.000, E1   -40.916, E3 +9635.439}
SPL {X  -159.990, Y  +405.475, Z    +0.000, E1   -51.039, E3 +9635.956}
SPL {X  -159.990, Y  +414.231, Z    +0.000, E1   -60.575, E3 +9637.140}
SPL {X  -159.990, Y  +462.953, Z    +0.000, E1   -73.611, E3 +9648.879}
SPL {X  -153.839, Y  +715.436, Z    +0.000, E1   -75.884, E3 +9751.310}
SPL {X  -148.840, Y  +730.182, Z    +0.000, E1   -75.434, E3 +9763.886}
SPL {X  -143.409, Y  +742.426, Z    +0.000, E1   -74.905, E3 +9775.398}
SPL {X  -139.557, Y  +749.735, Z    +0.000, E1   -74.483, E3 +9782.746}
SPL {X  -136.371, Y  +755.165, Z    +0.000, E1   -74.152, E3 +9788.292}
SPL {X  -133.102, Y  +760.274, Z    +0.000, E1   -73.777, E3 +9793.677}
SPL {X  -128.975, Y  +766.169, Z    +0.000, E1   -73.313, E3 +9799.952}
SPL {X  -124.947, Y  +771.425, Z    +0.000, E1   -72.782, E3 +9805.645}
SPL {X  -121.698, Y  +775.357, Z    +0.000, E1   -72.353, E3 +9809.840}
SPL {X  -118.622, Y  +778.858, Z    +0.000, E1   -71.924, E3 +9813.466}
SPL {X   -66.171, Y  +817.165, Z    +0.000, E1   -56.016, E3 +9964.824}
ENDSPLINE

SPLINE
SPL {X  -126.418, Y  +769.557, Z    +0.000, E1   -57.118, E3 +10148.065}
SPL {X  -145.244, Y  +738.589, Z    +0.000, E1   -50.405, E3 +10161.307}
SPL {X  -150.151, Y  +726.741, Z    +0.000, E1   -46.068, E3 +10164.234}
SPL {X  -156.642, Y  +704.059, Z    +0.000, E1   -33.659, E3 +10167.863}
SPL {X  -159.317, Y  +686.157, Z    +0.000, E1   -18.660, E3 +10169.353}
SPL {X  -159.973, Y  +673.799, Z    +0.000, E1    -5.345, E3 +10169.802}
SPL {X  -159.990, Y  +669.500, Z    +0.000, E1    +0.000, E3 +10169.842}
SPL {X  -159.990, Y  +667.794, Z    +0.000, E1    +4.255, E3 +10169.853}
SPL {X  -159.990, Y  +664.091, Z    +0.000, E1   +14.928, E3 +10169.925}
SPL {X  -159.990, Y  +659.599, Z    +0.000, E1   +28.016, E3 +10170.096}
SPL {X  -159.990, Y  +652.711, Z    +0.000, E1   +44.293, E3 +10170.575}
SPL {X  -159.990, Y  +640.730, Z    +0.000, E1   +60.297, E3 +10171.924}
SPL {X  -159.990, Y  +620.478, Z    +0.000, E1   +70.026, E3 +10175.738}
SPL {X  -159.990, Y  +573.021, Z    +0.000, E1   +74.619, E3 +10189.681}
SPL {X  -154.165, Y  +339.724, Z    +0.000, E1   +75.927, E3 +10285.528}
SPL {X  -150.571, Y  +328.416, Z    +0.000, E1   +75.599, E3 +10294.974}
SPL {X  -148.206, Y  +322.236, Z    +0.000, E1   +75.365, E3 +10300.518}
SPL {X  -136.549, Y  +299.126, Z    +0.000, E1   +77.537, E3 +10288.683}
ENDSPLINE

SPLINE
SPL {X  -136.862, Y  +299.641, Z    +0.000, E1   +76.604, E3 +10297.325}
ENDSPLINE

SPLINE
SPL {X  -136.434, Y  +298.938, Z    +0.000, E1   +75.982, E3 +10303.216}
SPL {X  -135.890, Y  +298.057, Z    +0.000, E1   +75.040, E3 +10311.682}
SPL {X  -134.349, Y  +295.626, Z    +0.000, E1   +74.322, E3 +10318.530}
SPL {X  -131.287, Y  +291.064, Z    +0.000, E1   +73.972, E3 +10323.342}
SPL {X  -128.265, Y  +286.871, Z    +0.000, E1   +73.613, E3 +10327.798}
SPL {X  -125.161, Y  +282.843, Z    +0.000, E1   +73.232, E3 +10332.070}
SPL {X  -122.038, Y  +279.042, Z    +0.000, E1   +72.832, E3 +10336.050}
SPL {X  -118.642, Y  +275.165, Z    +0.000, E1   +72.381, E3 +10340.013}
SPL {X   -66.040, Y  +236.776, Z    +0.000, E1   +55.694, E3 +10501.376}
ENDSPLINE

SPLINE
SPL {X  -127.452, Y  +285.790, Z    +0.000, E1   +56.591, E3 +10675.322}
SPL {X  -151.591, Y  +331.344, Z    +0.000, E1   +43.870, E3 +10691.421}
SPL {X  -158.135, Y  +358.205, Z    +0.000, E1   +26.984, E3 +10695.149}
SPL {X  -159.602, Y  +371.361, Z    +0.000, E1   +14.835, E3 +10696.045}
SPL {X  -159.981, Y  +380.818, Z    +0.000, E1    +4.512, E3 +10696.322}
SPL {X  -159.990, Y  +384.681, Z    +0.000, E1    -0.222, E3 +10696.351}
SPL {X  -159.990, Y  +387.626, Z    +0.000, E1    -8.190, E3 +10696.380}
SPL {X  -159.990, Y  +390.340, Z    +0.000, E1   -15.987, E3 +10696.444}
SPL {X  -159.990, Y  +394.216, Z    +0.000, E1   -27.062, E3 +10696.606}
SPL {X  -159.990, Y  +399.855, Z    +0.000, E1   -40.916, E3 +10696.977}
SPL {X  -159.990, Y  +405.475, Z    +0.000, E1   -51.039, E3 +10697.494}
SPL {X  -159.990, Y  +414.231, Z    +0.000, E1   -60.575, E3 +10698.678}
SPL {X  -159.990, Y  +462.953, Z    +0.000, E1   -73.611, E3 +10710.417}
SPL {X  -153.839, Y  +715.436, Z    +0.000, E1   -75.884, E3 +10812.848}
SPL {X  -148.840, Y  +730.182, Z    +0.000, E1   -75.434, E3 +10825.425}
SPL {X  -143.409, Y  +742.426, Z    +0.000, E1   -74.905, E3 +10836.937}
SPL {X  -139.557, Y  +749.735, Z    +0.000, E1   -74.483, E3 +10844.285}
SPL {X  -136.371, Y  +755.165, Z    +0.000, E1   -74.152, E3 +10849.830}
SPL {X  -133.102, Y  +760.274, Z    +0.000, E1   -73.777, E3 +10855.215}
SPL {X  -128.975, Y  +766.169, Z    +0.000, E1   -73.313, E3 +10861.491}
SPL {X  -124.947, Y  +771.425, Z    +0.000, E1   -72.782, E3 +10867.184}
SPL {X  -121.698, Y  +775.357, Z    +0.000, E1   -72.353, E3 +10871.378}
SPL {X  -118.622, Y  +778.858, Z    +0.000, E1   -71.924, E3 +10875.004}
SPL {X   -66.171, Y  +817.165, Z    +0.000, E1   -56.016, E3 +11026.363}
ENDSPLINE

SPLINE
SPL {X  -126.418, Y  +769.557, Z    +0.000, E1   -57.118, E3 +11209.604}
SPL {X  -148.476, Y  +731.097, Z    +0.000, E1   -47.824, E3 +11224.760}
SPL {X  -156.642, Y  +704.059, Z    +0.000, E1   -33.659, E3 +11229.402}
SPL {X  -159.317, Y  +686.157, Z    +0.000, E1   -18.660, E3 +11230.892}
SPL {X  -159.973, Y  +673.799, Z    +0.000, E1    -5.345, E3 +11231.340}
SPL {X  -159.990, Y  +669.500, Z    +0.000, E1    +0.000, E3 +11231.381}
SPL {X  -159.990, Y  +667.794, Z    +0.000, E1    +4.255, E3 +11231.392}
SPL {X  -159.990, Y  +664.091, Z    +0.000, E1   +14.928, E3 +11231.464}
SPL {X  -159.990, Y  +659.599, Z    +0.000, E1   +28.016, E3 +11231.634}
SPL {X  -159.990, Y  +652.711, Z    +0.000, E1   +44.293, E3 +11232.114}
SPL {X  -159.990, Y  +640.730, Z    +0.000, E1   +60.297, E3 +11233.463}
SPL {X  -159.990, Y  +620.478, Z    +0.000, E1   +70.026, E3 +11237.276}
SPL {X  -159.990, Y  +573.021, Z    +0.000, E1   +74.619, E3 +11251.220}
SPL {X  -154.165, Y  +339.724, Z    +0.000, E1   +75.927, E3 +11347.067}
SPL {X  -150.223, Y  +327.456, Z    +0.000, E1   +75.573, E3 +11357.332}
SPL {X  -136.549, Y  +299.126, Z    +0.000, E1   +77.537, E3 +11350.222}
ENDSPLINE

SPLINE
SPL {X  -136.862, Y  +299.641, Z    +0.000, E1   +76.604, E3 +11358.864}
ENDSPLINE

SPLINE
SPL {X  -136.434, Y  +298.938, Z    +0.000, E1   +75.982, E3 +11364.755}
SPL {X  -135.890, Y  +298.057, Z    +0.000, E1   +75.040, E3 +11373.221}
SPL {X  -134.349, Y  +295.626, Z    +0.000, E1   +74.322, E3 +11380.068}
SPL {X  -131.287, Y  +291.064, Z    +0.000, E1   +73.972, E3 +11384.881}
SPL {X  -128.265, Y  +286.871, Z    +0.000, E1   +73.613, E3 +11389.337}
SPL {X  -125.161, Y  +282.843, Z    +0.000, E1   +73.232, E3 +11393.608}
SPL {X  -122.038, Y  +279.042, Z    +0.000, E1   +72.832, E3 +11397.588}
SPL {X  -118.642, Y  +275.165, Z    +0.000, E1   +72.381, E3 +11401.551}
SPL {X   -66.040, Y  +236.776, Z    +0.000, E1   +55.694, E3 +11562.915}
ENDSPLINE

SPLINE
SPL {X  -127.452, Y  +285.790, Z    +0.000, E1   +56.591, E3 +11736.860}
SPL {X  -151.591, Y  +331.344, Z    +0.000, E1   +43.870, E3 +11752.959}
SPL {X  -158.135, Y  +358.205, Z    +0.000, E1   +26.984, E3 +11756.687}
SPL {X  -159.602, Y  +371.361, Z    +0.000, E1   +14.835, E3 +11757.583}
SPL {X  -159.981, Y  +380.818, Z    +0.000, E1    +4.512, E3 +11757.861}
SPL {X  -159.990, Y  +384.681, Z    +0.000, E1    -0.222, E3 +11757.890}
SPL {X  -159.990, Y  +387.626, Z    +0.000, E1    -8.190, E3 +11757.918}
SPL {X  -159.990, Y  +390.340, Z    +0.000, E1   -15.987, E3 +11757.983}
SPL {X  -159.990, Y  +394.216, Z    +0.000, E1   -27.062, E3 +11758.145}
SPL {X  -159.990, Y  +399.855, Z    +0.000, E1   -40.916, E3 +11758.516}
SPL {X  -159.990, Y  +405.475, Z    +0.000, E1   -51.039, E3 +11759.033}
SPL {X  -159.990, Y  +414.231, Z    +0.000, E1   -60.575, E3 +11760.217}
SPL {X  -159.990, Y  +462.953, Z    +0.000, E1   -73.611, E3 +11771.956}
SPL {X  -153.839, Y  +715.436, Z    +0.000, E1   -75.884, E3 +11874.386}
SPL {X  -148.840, Y  +730.182, Z    +0.000, E1   -75.434, E3 +11886.963}
SPL {X  -143.409, Y  +742.426, Z    +0.000, E1   -74.905, E3 +11898.475}
SPL {X  -139.557, Y  +749.735, Z    +0.000, E1   -74.483, E3 +11905.823}
SPL {X  -136.371, Y  +755.165, Z    +0.000, E1   -74.152, E3 +11911.369}
SPL {X  -133.102, Y  +760.274, Z    +0.000, E1   -73.777, E3 +11916.754}
SPL {X  -128.975, Y  +766.169, Z    +0.000, E1   -73.313, E3 +11923.029}
SPL {X  -124.947, Y  +771.425, Z    +0.000, E1   -72.782, E3 +11928.722}
SPL {X  -121.698, Y  +775.357, Z    +0.000, E1   -72.353, E3 +11932.917}
SPL {X  -118.622, Y  +778.858, Z    +0.000, E1   -71.924, E3 +11936.543}
SPL {X   -66.171, Y  +817.165, Z    +0.000, E1   -56.016, E3 +12087.901}
ENDSPLINE

SPLINE
SPL {X  -126.418, Y  +769.557, Z    +0.000, E1   -57.118, E3 +12271.142}
SPL {X  -148.476, Y  +731.097, Z    +0.000, E1   -47.824, E3 +12286.298}
SPL {X  -156.642, Y  +704.059, Z    +0.000, E1   -33.659, E3 +12290.940}
SPL {X  -159.317, Y  +686.157, Z    +0.000, E1   -18.660, E3 +12292.430}
SPL {X  -159.973, Y  +673.799, Z    +0.000, E1    -5.345, E3 +12292.879}
SPL {X  -159.990, Y  +669.500, Z    +0.000, E1    +0.000, E3 +12292.919}
SPL {X  -159.990, Y  +667.794, Z    +0.000, E1    +4.255, E3 +12292.930}
SPL {X  -159.990, Y  +664.091, Z    +0.000, E1   +14.928, E3 +12293.002}
SPL {X  -159.990, Y  +659.599, Z    +0.000, E1   +28.016, E3 +12293.173}
SPL {X  -159.990, Y  +652.711, Z    +0.000, E1   +44.293, E3 +12293.652}
SPL {X  -159.990, Y  +640.730, Z    +0.000, E1   +60.297, E3 +12295.001}
SPL {X  -159.990, Y  +620.478, Z    +0.000, E1   +70.026, E3 +12298.814}
SPL {X  -159.990, Y  +573.021, Z    +0.000, E1   +74.619, E3 +12312.758}
SPL {X  -154.165, Y  +339.724, Z    +0.000, E1   +75.927, E3 +12408.605}
SPL {X  -150.223, Y  +327.456, Z    +0.000, E1   +75.573, E3 +12418.870}
SPL {X  -136.549, Y  +299.126, Z    +0.000, E1   +77.537, E3 +12411.760}
ENDSPLINE

SPLINE
SPL {X  -136.862, Y  +299.641, Z    +0.000, E1   +76.604, E3 +12420.402}
ENDSPLINE

SPLINE
SPL {X  -136.434, Y  +298.938, Z    +0.000, E1   +75.982, E3 +12426.293}
SPL {X  -135.890, Y  +298.057, Z    +0.000, E1   +75.040, E3 +12434.759}
SPL {X  -134.349, Y  +295.626, Z    +0.000, E1   +74.322, E3 +12441.606}
SPL {X  -131.287, Y  +291.064, Z    +0.000, E1   +73.972, E3 +12446.419}
SPL {X  -128.265, Y  +286.871, Z    +0.000, E1   +73.613, E3 +12450.875}
SPL {X  -125.161, Y  +282.843, Z    +0.000, E1   +73.232, E3 +12455.147}
SPL {X  -122.038, Y  +279.042, Z    +0.000, E1   +72.832, E3 +12459.127}
SPL {X  -118.642, Y  +275.165, Z    +0.000, E1   +72.381, E3 +12463.090}
SPL {X   -66.040, Y  +236.776, Z    +0.000, E1   +55.694, E3 +12624.453}
ENDSPLINE

SPLINE
SPL {X  -127.452, Y  +285.790, Z    +0.000, E1   +56.591, E3 +12798.399}
SPL {X  -151.591, Y  +331.344, Z    +0.000, E1   +43.870, E3 +12814.498}
SPL {X  -158.135, Y  +358.205, Z    +0.000, E1   +26.984, E3 +12818.226}
SPL {X  -159.602, Y  +371.361, Z    +0.000, E1   +14.835, E3 +12819.122}
SPL {X  -159.981, Y  +380.818, Z    +0.000, E1    +4.512, E3 +12819.399}
SPL {X  -159.990, Y  +384.681, Z    +0.000, E1    -0.222, E3 +12819.428}
SPL {X  -159.990, Y  +387.626, Z    +0.000, E1    -8.190, E3 +12819.457}
SPL {X  -159.990, Y  +390.340, Z    +0.000, E1   -15.987, E3 +12819.521}
SPL {X  -159.990, Y  +394.216, Z    +0.000, E1   -27.062, E3 +12819.683}
SPL {X  -159.990, Y  +399.855, Z    +0.000, E1   -40.916, E3 +12820.054}
SPL {X  -159.990, Y  +405.475, Z    +0.000, E1   -51.039, E3 +12820.571}
SPL {X  -159.990, Y  +414.231, Z    +0.000, E1   -60.575, E3 +12821.755}
SPL {X  -159.990, Y  +462.953, Z    +0.000, E1   -73.611, E3 +12833.494}
SPL {X  -153.839, Y  +715.436, Z    +0.000, E1   -75.884, E3 +12935.925}
SPL {X  -148.840, Y  +730.182, Z    +0.000, E1   -75.434, E3 +12948.502}
SPL {X  -143.409, Y  +742.426, Z    +0.000, E1   -74.905, E3 +12960.014}
SPL {X  -139.557, Y  +749.735, Z    +0.000, E1   -74.483, E3 +12967.362}
SPL {X  -136.371, Y  +755.165, Z    +0.000, E1   -74.152, E3 +12972.907}
SPL {X  -133.102, Y  +760.274, Z    +0.000, E1   -73.777, E3 +12978.292}
SPL {X  -128.975, Y  +766.169, Z    +0.000, E1   -73.313, E3 +12984.568}
SPL {X  -124.947, Y  +771.425, Z    +0.000, E1   -72.782, E3 +12990.261}
SPL {X  -121.698, Y  +775.357, Z    +0.000, E1   -72.353, E3 +12994.455}
SPL {X  -118.622, Y  +778.858, Z    +0.000, E1   -71.924, E3 +12998.081}
SPL {X   -66.171, Y  +817.165, Z    +0.000, E1   -56.016, E3 +13149.440}
ENDSPLINE

SPLINE
SPL {X  -126.418, Y  +769.557, Z    +0.000, E1   -57.118, E3 +13332.681}
SPL {X  -148.476, Y  +731.097, Z    +0.000, E1   -47.824, E3 +13347.837}
SPL {X  -156.642, Y  +704.059, Z    +0.000, E1   -33.659, E3 +13352.479}
SPL {X  -159.317, Y  +686.157, Z    +0.000, E1   -18.660, E3 +13353.969}
SPL {X  -159.973, Y  +673.799, Z    +0.000, E1    -5.345, E3 +13354.417}
SPL {X  -159.990, Y  +669.500, Z    +0.000, E1    +0.000, E3 +13354.457}
SPL {X  -159.990, Y  +667.794, Z    +0.000, E1    +4.255, E3 +13354.469}
SPL {X  -159.990, Y  +664.091, Z    +0.000, E1   +14.928, E3 +13354.541}
SPL {X  -159.990, Y  +659.599, Z    +0.000, E1   +28.016, E3 +13354.711}
SPL {X  -159.990, Y  +652.711, Z    +0.000, E1   +44.293, E3 +13355.191}
SPL {X  -159.990, Y  +640.730, Z    +0.000, E1   +60.297, E3 +13356.540}
SPL {X  -159.990, Y  +620.478, Z    +0.000, E1   +70.026, E3 +13360.353}
SPL {X  -159.990, Y  +573.021, Z    +0.000, E1   +74.619, E3 +13374.297}
SPL {X  -154.165, Y  +339.724, Z    +0.000, E1   +75.927, E3 +13470.144}
SPL {X  -150.223, Y  +327.456, Z    +0.000, E1   +75.573, E3 +13480.409}
SPL {X  -136.549, Y  +299.126, Z    +0.000, E1   +77.537, E3 +13473.299}
ENDSPLINE

SPLINE
SPL {X  -136.862, Y  +299.641, Z    +0.000, E1   +76.604, E3 +13481.941}
ENDSPLINE

SPLINE
SPL {X  -136.434, Y  +298.938, Z    +0.000, E1   +75.982, E3 +13487.832}
SPL {X  -135.890, Y  +298.057, Z    +0.000, E1   +75.040, E3 +13496.298}
SPL {X  -134.349, Y  +295.626, Z    +0.000, E1   +74.322, E3 +13503.145}
SPL {X  -131.287, Y  +291.064, Z    +0.000, E1   +73.972, E3 +13507.957}
SPL {X  -128.265, Y  +286.871, Z    +0.000, E1   +73.613, E3 +13512.413}
SPL {X  -125.161, Y  +282.843, Z    +0.000, E1   +73.232, E3 +13516.685}
SPL {X  -122.038, Y  +279.042, Z    +0.000, E1   +72.832, E3 +13520.665}
SPL {X  -118.642, Y  +275.165, Z    +0.000, E1   +72.381, E3 +13524.628}
SPL {X   -66.040, Y  +236.776, Z    +0.000, E1   +55.694, E3 +13685.992}
ENDSPLINE

SPLINE
SPL {X  -127.452, Y  +285.790, Z    +0.000, E1   +56.591, E3 +13859.937}
SPL {X  -151.591, Y  +331.344, Z    +0.000, E1   +43.870, E3 +13876.036}
SPL {X  -158.135, Y  +358.205, Z    +0.000, E1   +26.984, E3 +13879.764}
SPL {X  -159.602, Y  +371.361, Z    +0.000, E1   +14.835, E3 +13880.660}
SPL {X  -159.981, Y  +380.818, Z    +0.000, E1    +4.512, E3 +13880.938}
SPL {X  -159.990, Y  +384.681, Z    +0.000, E1    -0.222, E3 +13880.967}
SPL {X  -159.990, Y  +387.626, Z    +0.000, E1    -8.190, E3 +13880.995}
SPL {X  -159.990, Y  +390.340, Z    +0.000, E1   -15.987, E3 +13881.060}
SPL {X  -159.990, Y  +394.216, Z    +0.000, E1   -27.062, E3 +13881.222}
SPL {X  -159.990, Y  +399.855, Z    +0.000, E1   -40.916, E3 +13881.593}
SPL {X  -159.990, Y  +405.475, Z    +0.000, E1   -51.039, E3 +13882.110}
SPL {X  -159.990, Y  +414.231, Z    +0.000, E1   -60.575, E3 +13883.294}
SPL {X  -159.990, Y  +462.953, Z    +0.000, E1   -73.611, E3 +13895.033}
SPL {X  -153.839, Y  +715.436, Z    +0.000, E1   -75.884, E3 +13997.463}
SPL {X  -149.923, Y  +727.355, Z    +0.000, E1   -75.515, E3 +14007.573}
SPL {X  -145.995, Y  +736.939, Z    +0.000, E1   -75.150, E3 +14016.308}
SPL {X  -141.012, Y  +747.080, Z    +0.000, E1   -74.661, E3 +14026.160}
SPL {X  -136.371, Y  +755.165, Z    +0.000, E1   -74.152, E3 +14034.446}
SPL {X  -133.102, Y  +760.274, Z    +0.000, E1   -73.777, E3 +14039.831}
SPL {X  -128.975, Y  +766.169, Z    +0.000, E1   -73.313, E3 +14046.106}
SPL {X  -124.947, Y  +771.425, Z    +0.000, E1   -72.782, E3 +14051.799}
SPL {X  -121.698, Y  +775.357, Z    +0.000, E1   -72.353, E3 +14055.994}
SPL {X  -118.622, Y  +778.858, Z    +0.000, E1   -71.924, E3 +14059.620}
SPL {X   -66.171, Y  +817.165, Z    +0.000, E1   -56.016, E3 +14210.978}
ENDSPLINE

SPLINE
SPL {X  -126.418, Y  +769.557, Z    +0.000, E1   -57.118, E3 +14394.219}
SPL {X  -148.476, Y  +731.097, Z    +0.000, E1   -47.824, E3 +14409.375}
SPL {X  -156.642, Y  +704.059, Z    +0.000, E1   -33.659, E3 +14414.017}
SPL {X  -159.317, Y  +686.157, Z    +0.000, E1   -18.660, E3 +14415.507}
SPL {X  -159.907, Y  +676.666, Z    +0.000, E1    -8.555, E3 +14415.905}
SPL {X  -159.990, Y  +669.586, Z    +0.000, E1    -0.216, E3 +14415.996}
SPL {X  -159.990, Y  +667.794, Z    +0.000, E1    +4.255, E3 +14416.007}
SPL {X  -159.990, Y  +664.091, Z    +0.000, E1   +14.928, E3 +14416.079}
SPL {X  -159.990, Y  +659.599, Z    +0.000, E1   +28.016, E3 +14416.250}
SPL {X  -159.990, Y  +652.711, Z    +0.000, E1   +44.293, E3 +14416.729}
SPL {X  -159.990, Y  +640.730, Z    +0.000, E1   +60.297, E3 +14418.078}
SPL {X  -159.990, Y  +620.478, Z    +0.000, E1   +70.026, E3 +14421.891}
SPL {X  -159.990, Y  +573.021, Z    +0.000, E1   +74.619, E3 +14435.835}
SPL {X  -154.165, Y  +339.724, Z    +0.000, E1   +75.927, E3 +14531.682}
SPL {X  -150.223, Y  +327.456, Z    +0.000, E1   +75.573, E3 +14541.947}
SPL {X  -136.549, Y  +299.126, Z    +0.000, E1   +77.537, E3 +14534.837}
ENDSPLINE

SPLINE
SPL {X  -136.862, Y  +299.641, Z    +0.000, E1   +76.604, E3 +14543.479}
ENDSPLINE

SPLINE
SPL {X  -136.434, Y  +298.938, Z    +0.000, E1   +75.982, E3 +14549.370}
SPL {X  -135.890, Y  +298.057, Z    +0.000, E1   +75.040, E3 +14557.836}
SPL {X  -134.349, Y  +295.626, Z    +0.000, E1   +74.322, E3 +14564.683}
SPL {X  -131.287, Y  +291.064, Z    +0.000, E1   +73.972, E3 +14569.496}
SPL {X  -128.265, Y  +286.871, Z    +0.000, E1   +73.613, E3 +14573.952}
SPL {X  -125.161, Y  +282.843, Z    +0.000, E1   +73.232, E3 +14578.224}
SPL {X  -122.038, Y  +279.042, Z    +0.000, E1   +72.832, E3 +14582.204}
SPL {X  -118.642, Y  +275.165, Z    +0.000, E1   +72.381, E3 +14586.167}
SPL {X   -66.040, Y  +236.776, Z    +0.000, E1   +55.694, E3 +14747.530}
ENDSPLINE

SPLINE
SPL {X  -127.452, Y  +285.790, Z    +0.000, E1   +56.591, E3 +14921.476}
SPL {X  -148.001, Y  +321.733, Z    +0.000, E1   +47.810, E3 +14935.579}
SPL {X  -154.604, Y  +341.337, Z    +0.000, E1   +38.630, E3 +14939.353}
SPL {X  -158.135, Y  +358.205, Z    +0.000, E1   +26.984, E3 +14941.302}
SPL {X  -159.602, Y  +371.361, Z    +0.000, E1   +14.835, E3 +14942.198}
SPL {X  -159.981, Y  +380.818, Z    +0.000, E1    +4.512, E3 +14942.476}
SPL {X  -159.990, Y  +384.681, Z    +0.000, E1    -0.222, E3 +14942.505}
SPL {X  -159.990, Y  +389.079, Z    +0.000, E1   -12.017, E3 +14942.568}
SPL {X  -159.990, Y  +394.216, Z    +0.000, E1   -27.062, E3 +14942.760}
SPL {X  -159.990, Y  +399.855, Z    +0.000, E1   -40.916, E3 +14943.131}
SPL {X  -159.990, Y  +405.475, Z    +0.000, E1   -51.039, E3 +14943.648}
SPL {X  -159.990, Y  +414.231, Z    +0.000, E1   -60.575, E3 +14944.832}
SPL {X  -159.990, Y  +462.953, Z    +0.000, E1   -73.611, E3 +14956.571}
SPL {X  -153.839, Y  +715.436, Z    +0.000, E1   -75.884, E3 +15059.002}
SPL {X  -148.840, Y  +730.182, Z    +0.000, E1   -75.434, E3 +15071.578}
SPL {X  -143.409, Y  +742.426, Z    +0.000, E1   -74.905, E3 +15083.090}
SPL {X  -139.557, Y  +749.735, Z    +0.000, E1   -74.483, E3 +15090.439}
SPL {X  -136.371, Y  +755.165, Z    +0.000, E1   -74.152, E3 +15095.984}
SPL {X  -133.102, Y  +760.274, Z    +0.000, E1   -73.777, E3 +15101.369}
SPL {X  -128.975, Y  +766.169, Z    +0.000, E1   -73.313, E3 +15107.645}
SPL {X  -124.947, Y  +771.425, Z    +0.000, E1   -72.782, E3 +15113.338}
SPL {X  -121.698, Y  +775.357, Z    +0.000, E1   -72.353, E3 +15117.532}
SPL {X  -118.622, Y  +778.858, Z    +0.000, E1   -71.924, E3 +15121.158}
SPL {X   -66.171, Y  +817.165, Z    +0.000, E1   -56.016, E3 +15272.517}
ENDSPLINE

SPLINE
SPL {X  -126.418, Y  +769.557, Z    +0.000, E1   -57.118, E3 +15455.758}
SPL {X  -145.244, Y  +738.589, Z    +0.000, E1   -50.405, E3 +15468.999}
SPL {X  -150.151, Y  +726.741, Z    +0.000, E1   -46.068, E3 +15471.926}
SPL {X  -156.642, Y  +704.059, Z    +0.000, E1   -33.659, E3 +15475.555}
SPL {X  -159.317, Y  +686.157, Z    +0.000, E1   -18.660, E3 +15477.046}
SPL {X  -159.973, Y  +673.799, Z    +0.000, E1    -5.345, E3 +15477.494}
SPL {X  -159.990, Y  +669.500, Z    +0.000, E1    +0.000, E3 +15477.534}
SPL {X  -159.990, Y  +667.794, Z    +0.000, E1    +4.255, E3 +15477.546}
SPL {X  -159.990, Y  +664.091, Z    +0.000, E1   +14.928, E3 +15477.618}
SPL {X  -159.990, Y  +658.301, Z    +0.000, E1   +31.283, E3 +15477.870}
SPL {X  -159.990, Y  +650.845, Z    +0.000, E1   +47.892, E3 +15478.415}
SPL {X  -159.990, Y  +640.730, Z    +0.000, E1   +60.297, E3 +15479.617}
SPL {X  -159.990, Y  +620.478, Z    +0.000, E1   +70.026, E3 +15483.430}
SPL {X  -159.990, Y  +573.021, Z    +0.000, E1   +74.619, E3 +15497.374}
SPL {X  -154.165, Y  +339.724, Z    +0.000, E1   +75.927, E3 +15593.221}
SPL {X  -150.223, Y  +327.456, Z    +0.000, E1   +75.573, E3 +15603.486}
SPL {X  -136.549, Y  +299.126, Z    +0.000, E1   +77.537, E3 +15596.376}
ENDSPLINE

SPLINE
SPL {X  -136.862, Y  +299.641, Z    +0.000, E1   +76.604, E3 +15605.018}
ENDSPLINE

SPLINE
SPL {X  -136.434, Y  +298.938, Z    +0.000, E1   +75.982, E3 +15610.909}
SPL {X  -135.890, Y  +298.057, Z    +0.000, E1   +75.040, E3 +15619.375}
SPL {X  -134.349, Y  +295.626, Z    +0.000, E1   +74.322, E3 +15626.222}
SPL {X  -131.287, Y  +291.064, Z    +0.000, E1   +73.972, E3 +15631.034}
SPL {X  -128.265, Y  +286.871, Z    +0.000, E1   +73.613, E3 +15635.490}
SPL {X  -125.161, Y  +282.843, Z    +0.000, E1   +73.232, E3 +15639.762}
SPL {X  -122.038, Y  +279.042, Z    +0.000, E1   +72.832, E3 +15643.742}
SPL {X  -118.642, Y  +275.165, Z    +0.000, E1   +72.381, E3 +15647.705}
SPL {X   -66.040, Y  +236.776, Z    +0.000, E1   +55.694, E3 +15809.069}
ENDSPLINE

SPLINE
SPL {X  -127.452, Y  +285.790, Z    +0.000, E1   +56.591, E3 +15983.014}
SPL {X  -151.591, Y  +331.344, Z    +0.000, E1   +43.870, E3 +15999.113}
SPL {X  -158.135, Y  +358.205, Z    +0.000, E1   +26.984, E3 +16002.841}
SPL {X  -159.602, Y  +371.361, Z    +0.000, E1   +14.835, E3 +16003.737}
SPL {X  -159.981, Y  +380.818, Z    +0.000, E1    +4.512, E3 +16004.015}
SPL {X  -159.990, Y  +384.681, Z    +0.000, E1    -0.222, E3 +16004.044}
SPL {X  -159.990, Y  +387.626, Z    +0.000, E1    -8.190, E3 +16004.072}
SPL {X  -159.990, Y  +390.340, Z    +0.000, E1   -15.987, E3 +16004.137}
SPL {X  -159.990, Y  +394.216, Z    +0.000, E1   -27.062, E3 +16004.299}
SPL {X  -159.990, Y  +399.855, Z    +0.000, E1   -40.916, E3 +16004.670}
SPL {X  -159.990, Y  +405.475, Z    +0.000, E1   -51.039, E3 +16005.187}
SPL {X  -159.990, Y  +414.231, Z    +0.000, E1   -60.575, E3 +16006.371}
SPL {X  -159.990, Y  +462.953, Z    +0.000, E1   -73.611, E3 +16018.110}
SPL {X  -153.839, Y  +715.436, Z    +0.000, E1   -75.884, E3 +16120.540}
SPL {X  -149.923, Y  +727.355, Z    +0.000, E1   -75.515, E3 +16130.650}
SPL {X  -145.995, Y  +736.939, Z    +0.000, E1   -75.150, E3 +16139.385}
SPL {X  -141.012, Y  +747.080, Z    +0.000, E1   -74.661, E3 +16149.237}
SPL {X  -136.371, Y  +755.165, Z    +0.000, E1   -74.152, E3 +16157.523}
SPL {X  -131.455, Y  +762.694, Z    +0.000, E1   -73.615, E3 +16165.441}
SPL {X  -125.933, Y  +770.180, Z    +0.000, E1   -72.934, E3 +16173.505}
SPL {X  -121.698, Y  +775.357, Z    +0.000, E1   -72.353, E3 +16179.071}
SPL {X  -118.622, Y  +778.858, Z    +0.000, E1   -71.924, E3 +16182.697}
SPL {X   -66.171, Y  +817.165, Z    +0.000, E1   -56.016, E3 +16334.055}
ENDSPLINE

SPLINE
SPL {X  -126.418, Y  +769.557, Z    +0.000, E1   -57.118, E3 +16517.296}
SPL {X  -145.244, Y  +738.589, Z    +0.000, E1   -50.405, E3 +16530.538}
SPL {X  -150.151, Y  +726.741, Z    +0.000, E1   -46.068, E3 +16533.464}
SPL {X  -156.642, Y  +704.059, Z    +0.000, E1   -33.659, E3 +16537.094}
SPL {X  -159.317, Y  +686.157, Z    +0.000, E1   -18.660, E3 +16538.584}
SPL {X  -159.973, Y  +673.799, Z    +0.000, E1    -5.345, E3 +16539.033}
SPL {X  -159.990, Y  +669.500, Z    +0.000, E1    +0.000, E3 +16539.073}
SPL {X  -159.990, Y  +667.794, Z    +0.000, E1    +4.255, E3 +16539.084}
SPL {X  -159.990, Y  +664.091, Z    +0.000, E1   +14.928, E3 +16539.156}
SPL {X  -159.990, Y  +658.301, Z    +0.000, E1   +31.283, E3 +16539.409}
SPL {X  -159.990, Y  +650.845, Z    +0.000, E1   +47.892, E3 +16539.954}
SPL {X  -159.990, Y  +640.730, Z    +0.000, E1   +60.297, E3 +16541.155}
SPL {X  -159.990, Y  +620.478, Z    +0.000, E1   +70.026, E3 +16544.968}
SPL {X  -159.990, Y  +573.021, Z    +0.000, E1   +74.619, E3 +16558.912}
SPL {X  -154.165, Y  +339.724, Z    +0.000, E1   +75.927, E3 +16654.759}
SPL {X  -150.223, Y  +327.456, Z    +0.000, E1   +75.573, E3 +16665.024}
SPL {X  -136.549, Y  +299.126, Z    +0.000, E1   +77.537, E3 +16657.914}
ENDSPLINE

SPLINE
SPL {X  -136.862, Y  +299.641, Z    +0.000, E1   +76.604, E3 +16666.556}
ENDSPLINE

SPLINE
SPL {X  -136.434, Y  +298.938, Z    +0.000, E1   +75.982, E3 +16672.447}
SPL {X  -135.890, Y  +298.057, Z    +0.000, E1   +75.040, E3 +16680.913}
SPL {X  -134.349, Y  +295.626, Z    +0.000, E1   +74.322, E3 +16687.760}
SPL {X  -131.287, Y  +291.064, Z    +0.000, E1   +73.972, E3 +16692.573}
SPL {X  -128.265, Y  +286.871, Z    +0.000, E1   +73.613, E3 +16697.029}
SPL {X  -125.161, Y  +282.843, Z    +0.000, E1   +73.232, E3 +16701.301}
SPL {X  -122.038, Y  +279.042, Z    +0.000, E1   +72.832, E3 +16705.281}
SPL {X  -118.642, Y  +275.165, Z    +0.000, E1   +72.381, E3 +16709.244}
SPL {X   -66.040, Y  +236.776, Z    +0.000, E1   +55.694, E3 +16870.607}
ENDSPLINE

SPLINE
SPL {X  -127.452, Y  +285.790, Z    +0.000, E1   +56.591, E3 +17044.552}
SPL {X  -151.591, Y  +331.344, Z    +0.000, E1   +43.870, E3 +17060.652}
SPL {X  -158.135, Y  +358.205, Z    +0.000, E1   +26.984, E3 +17064.379}
SPL {X  -159.602, Y  +371.361, Z    +0.000, E1   +14.835, E3 +17065.275}
SPL {X  -159.981, Y  +380.818, Z    +0.000, E1    +4.512, E3 +17065.553}
SPL {X  -159.990, Y  +384.681, Z    +0.000, E1    -0.222, E3 +17065.582}
SPL {X  -159.990, Y  +387.626, Z    +0.000, E1    -8.190, E3 +17065.611}
SPL {X  -159.990, Y  +390.340, Z    +0.000, E1   -15.987, E3 +17065.675}
SPL {X  -159.990, Y  +394.216, Z    +0.000, E1   -27.062, E3 +17065.837}
SPL {X  -159.990, Y  +399.855, Z    +0.000, E1   -40.916, E3 +17066.208}
SPL {X  -159.990, Y  +405.475, Z    +0.000, E1   -51.039, E3 +17066.725}
SPL {X  -159.990, Y  +414.231, Z    +0.000, E1   -60.575, E3 +17067.909}
SPL {X  -159.990, Y  +462.953, Z    +0.000, E1   -73.611, E3 +17079.648}
SPL {X  -153.839, Y  +715.436, Z    +0.000, E1   -75.884, E3 +17182.079}
SPL {X  -148.840, Y  +730.182, Z    +0.000, E1   -75.434, E3 +17194.655}
SPL {X  -143.409, Y  +742.426, Z    +0.000, E1   -74.905, E3 +17206.167}
SPL {X  -139.557, Y  +749.735, Z    +0.000, E1   -74.483, E3 +17213.515}
SPL {X  -136.371, Y  +755.165, Z    +0.000, E1   -74.152, E3 +17219.061}
SPL {X  -133.102, Y  +760.274, Z    +0.000, E1   -73.777, E3 +17224.446}
SPL {X  -128.975, Y  +766.169, Z    +0.000, E1   -73.313, E3 +17230.722}
SPL {X  -124.947, Y  +771.425, Z    +0.000, E1   -72.782, E3 +17236.415}
SPL {X  -121.698, Y  +775.357, Z    +0.000, E1   -72.353, E3 +17240.609}
SPL {X  -118.622, Y  +778.858, Z    +0.000, E1   -71.924, E3 +17244.235}
SPL {X   -66.171, Y  +817.165, Z    +0.000, E1   -56.016, E3 +17395.593}
ENDSPLINE

SPLINE
SPL {X  -126.418, Y  +769.557, Z    +0.000, E1   -57.118, E3 +17578.835}
SPL {X  -145.244, Y  +738.589, Z    +0.000, E1   -50.405, E3 +17592.076}
SPL {X  -150.151, Y  +726.741, Z    +0.000, E1   -46.068, E3 +17595.003}
SPL {X  -156.642, Y  +704.059, Z    +0.000, E1   -33.659, E3 +17598.632}
SPL {X  -159.317, Y  +686.157, Z    +0.000, E1   -18.660, E3 +17600.123}
SPL {X  -159.973, Y  +673.799, Z    +0.000, E1    -5.345, E3 +17600.571}
SPL {X  -159.990, Y  +669.500, Z    +0.000, E1    +0.000, E3 +17600.611}
SPL {X  -159.990, Y  +667.794, Z    +0.000, E1    +4.255, E3 +17600.623}
SPL {X  -159.990, Y  +664.091, Z    +0.000, E1   +14.928, E3 +17600.695}
SPL {X  -159.990, Y  +659.599, Z    +0.000, E1   +28.016, E3 +17600.865}
SPL {X  -159.990, Y  +652.711, Z    +0.000, E1   +44.293, E3 +17601.344}
SPL {X  -159.990, Y  +640.730, Z    +0.000, E1   +60.297, E3 +17602.693}
SPL {X  -159.990, Y  +620.478, Z    +0.000, E1   +70.026, E3 +17606.507}
SPL {X  -159.990, Y  +573.021, Z    +0.000, E1   +74.619, E3 +17620.451}
SPL {X  -154.165, Y  +339.724, Z    +0.000, E1   +75.927, E3 +17716.298}
SPL {X  -150.571, Y  +328.416, Z    +0.000, E1   +75.599, E3 +17725.743}
SPL {X  -148.206, Y  +322.236, Z    +0.000, E1   +75.365, E3 +17731.287}
SPL {X  -136.549, Y  +299.126, Z    +0.000, E1   +77.537, E3 +17719.452}
ENDSPLINE

SPLINE
SPL {X  -136.862, Y  +299.641, Z    +0.000, E1   +76.604, E3 +17728.094}
ENDSPLINE

SPLINE
SPL {X  -136.434, Y  +298.938, Z    +0.000, E1   +75.982, E3 +17733.986}
SPL {X  -135.890, Y  +298.057, Z    +0.000, E1   +75.040, E3 +17742.452}
SPL {X  -134.349, Y  +295.626, Z    +0.000, E1   +74.322, E3 +17749.299}
SPL {X  -131.287, Y  +291.064, Z    +0.000, E1   +73.972, E3 +17754.111}
SPL {X  -128.265, Y  +286.871, Z    +0.000, E1   +73.613, E3 +17758.567}
SPL {X  -125.161, Y  +282.843, Z    +0.000, E1   +73.232, E3 +17762.839}
SPL {X  -122.038, Y  +279.042, Z    +0.000, E1   +72.832, E3 +17766.819}
SPL {X  -118.642, Y  +275.165, Z    +0.000, E1   +72.381, E3 +17770.782}
SPL {X   -66.040, Y  +236.776, Z    +0.000, E1   +55.694, E3 +17932.146}
ENDSPLINE

SPLINE
SPL {X  -127.452, Y  +285.790, Z    +0.000, E1   +56.591, E3 +18106.091}
SPL {X  -151.591, Y  +331.344, Z    +0.000, E1   +43.870, E3 +18122.190}
SPL {X  -158.135, Y  +358.205, Z    +0.000, E1   +26.984, E3 +18125.918}
SPL {X  -159.602, Y  +371.361, Z    +0.000, E1   +14.835, E3 +18126.814}
SPL {X  -159.981, Y  +380.818, Z    +0.000, E1    +4.512, E3 +18127.092}
SPL {X  -159.990, Y  +384.681, Z    +0.000, E1    -0.222, E3 +18127.121}
SPL {X  -159.990, Y  +387.626, Z    +0.000, E1    -8.190, E3 +18127.149}
SPL {X  -159.990, Y  +390.340, Z    +0.000, E1   -15.987, E3 +18127.214}
SPL {X  -159.990, Y  +394.216, Z    +0.000, E1   -27.062, E3 +18127.375}
SPL {X  -159.990, Y  +399.855, Z    +0.000, E1   -40.916, E3 +18127.747}
SPL {X  -159.990, Y  +405.475, Z    +0.000, E1   -51.039, E3 +18128.263}
SPL {X  -159.990, Y  +414.231, Z    +0.000, E1   -60.575, E3 +18129.448}
SPL {X  -159.990, Y  +462.953, Z    +0.000, E1   -73.611, E3 +18141.187}
SPL {X  -153.839, Y  +715.436, Z    +0.000, E1   -75.884, E3 +18243.617}
SPL {X  -148.840, Y  +730.182, Z    +0.000, E1   -75.434, E3 +18256.194}
SPL {X  -143.409, Y  +742.426, Z    +0.000, E1   -74.905, E3 +18267.706}
SPL {X  -139.557, Y  +749.735, Z    +0.000, E1   -74.483, E3 +18275.054}
SPL {X  -136.371, Y  +755.165, Z    +0.000, E1   -74.152, E3 +18280.600}
SPL {X  -133.102, Y  +760.274, Z    +0.000, E1   -73.777, E3 +18285.985}
SPL {X  -128.975, Y  +766.169, Z    +0.000, E1   -73.313, E3 +18292.260}
SPL {X  -124.947, Y  +771.425, Z    +0.000, E1   -72.782, E3 +18297.953}
SPL {X  -121.698, Y  +775.357, Z    +0.000, E1   -72.353, E3 +18302.148}
SPL {X  -118.622, Y  +778.858, Z    +0.000, E1   -71.924, E3 +18305.774}
SPL {X   -66.171, Y  +817.165, Z    +0.000, E1   -56.016, E3 +18457.132}
ENDSPLINE

SPLINE
SPL {X  -126.418, Y  +769.557, Z    +0.000, E1   -57.118, E3 +18640.373}
SPL {X  -148.476, Y  +731.097, Z    +0.000, E1   -47.824, E3 +18655.529}
SPL {X  -156.642, Y  +704.059, Z    +0.000, E1   -33.659, E3 +18660.171}
SPL {X  -159.317, Y  +686.157, Z    +0.000, E1   -18.660, E3 +18661.661}
SPL {X  -159.973, Y  +673.799, Z    +0.000, E1    -5.345, E3 +18662.110}
SPL {X  -159.990, Y  +669.500, Z    +0.000, E1    +0.000, E3 +18662.150}
SPL {X  -159.990, Y  +667.794, Z    +0.000, E1    +4.255, E3 +18662.161}
SPL {X  -159.990, Y  +664.091, Z    +0.000, E1   +14.928, E3 +18662.233}
SPL {X  -159.990, Y  +659.599, Z    +0.000, E1   +28.016, E3 +18662.404}
SPL {X  -159.990, Y  +652.711, Z    +0.000, E1   +44.293, E3 +18662.883}
SPL {X  -159.990, Y  +640.730, Z    +0.000, E1   +60.297, E3 +18664.232}
SPL {X  -159.990, Y  +620.478, Z    +0.000, E1   +70.026, E3 +18668.045}
SPL {X  -159.990, Y  +573.021, Z    +0.000, E1   +74.619, E3 +18681.989}
SPL {X  -154.165, Y  +339.724, Z    +0.000, E1   +75.927, E3 +18777.836}
SPL {X  -150.223, Y  +327.456, Z    +0.000, E1   +75.573, E3 +18788.101}
SPL {X  -136.549, Y  +299.126, Z    +0.000, E1   +77.537, E3 +18780.991}
ENDSPLINE

SPLINE
SPL {X  -136.862, Y  +299.641, Z    +0.000, E1   +76.604, E3 +18789.633}
ENDSPLINE

SPLINE
SPL {X  -136.434, Y  +298.938, Z    +0.000, E1   +75.982, E3 +18795.524}
SPL {X  -135.890, Y  +298.057, Z    +0.000, E1   +75.040, E3 +18803.990}
SPL {X  -134.349, Y  +295.626, Z    +0.000, E1   +74.322, E3 +18810.837}
SPL {X  -131.287, Y  +291.064, Z    +0.000, E1   +73.972, E3 +18815.650}
SPL {X  -128.265, Y  +286.871, Z    +0.000, E1   +73.613, E3 +18820.106}
SPL {X  -125.161, Y  +282.843, Z    +0.000, E1   +73.232, E3 +18824.378}
SPL {X  -122.038, Y  +279.042, Z    +0.000, E1   +72.832, E3 +18828.357}
SPL {X  -118.642, Y  +275.165, Z    +0.000, E1   +72.381, E3 +18832.321}
SPL {X   -66.040, Y  +236.776, Z    +0.000, E1   +55.694, E3 +18993.684}
ENDSPLINE

SPLINE
SPL {X  -127.452, Y  +285.790, Z    +0.000, E1   +56.591, E3 +19167.629}
SPL {X  -151.591, Y  +331.344, Z    +0.000, E1   +43.870, E3 +19183.729}
SPL {X  -158.135, Y  +358.205, Z    +0.000, E1   +26.984, E3 +19187.456}
SPL {X  -159.602, Y  +371.361, Z    +0.000, E1   +14.835, E3 +19188.352}
SPL {X  -159.981, Y  +380.818, Z    +0.000, E1    +4.512, E3 +19188.630}
SPL {X  -159.990, Y  +384.681, Z    +0.000, E1    -0.222, E3 +19188.659}
SPL {X  -159.990, Y  +387.626, Z    +0.000, E1    -8.190, E3 +19188.687}
SPL {X  -159.990, Y  +390.340, Z    +0.000, E1   -15.987, E3 +19188.752}
SPL {X  -159.990, Y  +394.216, Z    +0.000, E1   -27.062, E3 +19188.914}
SPL {X  -159.990, Y  +399.855, Z    +0.000, E1   -40.916, E3 +19189.285}
SPL {X  -159.990, Y  +405.475, Z    +0.000, E1   -51.039, E3 +19189.802}
SPL {X  -159.990, Y  +414.231, Z    +0.000, E1   -60.575, E3 +19190.986}
SPL {X  -159.990, Y  +462.953, Z    +0.000, E1   -73.611, E3 +19202.725}
SPL {X  -153.839, Y  +715.436, Z    +0.000, E1   -75.884, E3 +19305.156}
SPL {X  -148.840, Y  +730.182, Z    +0.000, E1   -75.434, E3 +19317.732}
SPL {X  -143.409, Y  +742.426, Z    +0.000, E1   -74.905, E3 +19329.244}
SPL {X  -139.557, Y  +749.735, Z    +0.000, E1   -74.483, E3 +19336.592}
SPL {X  -136.371, Y  +755.165, Z    +0.000, E1   -74.152, E3 +19342.138}
SPL {X  -133.102, Y  +760.274, Z    +0.000, E1   -73.777, E3 +19347.523}
SPL {X  -128.975, Y  +766.169, Z    +0.000, E1   -73.313, E3 +19353.799}
SPL {X  -124.947, Y  +771.425, Z    +0.000, E1   -72.782, E3 +19359.492}
SPL {X  -121.698, Y  +775.357, Z    +0.000, E1   -72.353, E3 +19363.686}
SPL {X  -118.622, Y  +778.858, Z    +0.000, E1   -71.924, E3 +19367.312}
SPL {X   -66.171, Y  +817.165, Z    +0.000, E1   -56.016, E3 +19518.670}
ENDSPLINE

SPLINE
SPL {X  -126.418, Y  +769.557, Z    +0.000, E1   -57.118, E3 +19701.912}
SPL {X  -148.476, Y  +731.097, Z    +0.000, E1   -47.824, E3 +19717.068}
SPL {X  -156.642, Y  +704.059, Z    +0.000, E1   -33.659, E3 +19721.709}
SPL {X  -159.317, Y  +686.157, Z    +0.000, E1   -18.660, E3 +19723.200}
SPL {X  -159.973, Y  +673.799, Z    +0.000, E1    -5.345, E3 +19723.648}
SPL {X  -159.990, Y  +669.500, Z    +0.000, E1    +0.000, E3 +19723.688}
SPL {X  -159.990, Y  +667.794, Z    +0.000, E1    +4.255, E3 +19723.699}
SPL {X  -159.990, Y  +664.091, Z    +0.000, E1   +14.928, E3 +19723.772}
SPL {X  -159.990, Y  +659.599, Z    +0.000, E1   +28.016, E3 +19723.942}
SPL {X  -159.990, Y  +652.711, Z    +0.000, E1   +44.293, E3 +19724.421}
SPL {X  -159.990, Y  +640.730, Z    +0.000, E1   +60.297, E3 +19725.770}
SPL {X  -159.990, Y  +620.478, Z    +0.000, E1   +70.026, E3 +19729.584}
SPL {X  -159.990, Y  +573.021, Z    +0.000, E1   +74.619, E3 +19743.528}
SPL {X  -154.165, Y  +339.724, Z    +0.000, E1   +75.927, E3 +19839.374}
SPL {X  -150.223, Y  +327.456, Z    +0.000, E1   +75.573, E3 +19849.639}
SPL {X  -136.549, Y  +299.126, Z    +0.000, E1   +77.537, E3 +19842.529}
ENDSPLINE

SPLINE
SPL {X  -136.862, Y  +299.641, Z    +0.000, E1   +76.604, E3 +19851.171}
ENDSPLINE

SPLINE
SPL {X  -136.434, Y  +298.938, Z    +0.000, E1   +75.982, E3 +19857.062}
SPL {X  -135.890, Y  +298.057, Z    +0.000, E1   +75.040, E3 +19865.528}
SPL {X  -134.349, Y  +295.626, Z    +0.000, E1   +74.322, E3 +19872.376}
SPL {X  -131.287, Y  +291.064, Z    +0.000, E1   +73.972, E3 +19877.188}
SPL {X  -128.265, Y  +286.871, Z    +0.000, E1   +73.613, E3 +19881.644}
SPL {X  -125.161, Y  +282.843, Z    +0.000, E1   +73.232, E3 +19885.916}
SPL {X  -122.038, Y  +279.042, Z    +0.000, E1   +72.832, E3 +19889.896}
SPL {X  -118.642, Y  +275.165, Z    +0.000, E1   +72.381, E3 +19893.859}
SPL {X   -66.040, Y  +236.776, Z    +0.000, E1   +55.694, E3 +20055.223}
ENDSPLINE

SPLINE
SPL {X  -127.452, Y  +285.790, Z    +0.000, E1   +56.591, E3 +20229.168}
SPL {X  -151.591, Y  +331.344, Z    +0.000, E1   +43.870, E3 +20245.267}
SPL {X  -158.135, Y  +358.205, Z    +0.000, E1   +26.984, E3 +20248.995}
SPL {X  -159.602, Y  +371.361, Z    +0.000, E1   +14.835, E3 +20249.891}
SPL {X  -159.981, Y  +380.818, Z    +0.000, E1    +4.512, E3 +20250.169}
SPL {X  -159.990, Y  +384.681, Z    +0.000, E1    -0.222, E3 +20250.198}
SPL {X  -159.990, Y  +387.626, Z    +0.000, E1    -8.190, E3 +20250.226}
SPL {X  -159.990, Y  +390.340, Z    +0.000, E1   -15.987, E3 +20250.290}
SPL {X  -159.990, Y  +394.216, Z    +0.000, E1   -27.062, E3 +20250.452}
SPL {X  -159.990, Y  +399.855, Z    +0.000, E1   -40.916, E3 +20250.823}
SPL {X  -159.990, Y  +405.475, Z    +0.000, E1   -51.039, E3 +20251.340}
SPL {X  -159.990, Y  +414.231, Z    +0.000, E1   -60.575, E3 +20252.525}
SPL {X  -159.990, Y  +462.953, Z    +0.000, E1   -73.611, E3 +20264.264}
SPL {X  -153.839, Y  +715.436, Z    +0.000, E1   -75.884, E3 +20366.694}
SPL {X  -148.840, Y  +730.182, Z    +0.000, E1   -75.434, E3 +20379.271}
SPL {X  -143.409, Y  +742.426, Z    +0.000, E1   -74.905, E3 +20390.783}
SPL {X  -139.557, Y  +749.735, Z    +0.000, E1   -74.483, E3 +20398.131}
SPL {X  -136.371, Y  +755.165, Z    +0.000, E1   -74.152, E3 +20403.677}
SPL {X  -133.102, Y  +760.274, Z    +0.000, E1   -73.777, E3 +20409.062}
SPL {X  -128.975, Y  +766.169, Z    +0.000, E1   -73.313, E3 +20415.337}
SPL {X  -124.947, Y  +771.425, Z    +0.000, E1   -72.782, E3 +20421.030}
SPL {X  -121.698, Y  +775.357, Z    +0.000, E1   -72.353, E3 +20425.225}
SPL {X  -118.622, Y  +778.858, Z    +0.000, E1   -71.924, E3 +20428.851}
SPL {X   -66.171, Y  +817.165, Z    +0.000, E1   -56.016, E3 +20580.209}
ENDSPLINE

SPLINE
SPL {X  -126.418, Y  +769.557, Z    +0.000, E1   -57.118, E3 +20763.450}
SPL {X  -148.476, Y  +731.097, Z    +0.000, E1   -47.824, E3 +20778.606}
SPL {X  -156.642, Y  +704.059, Z    +0.000, E1   -33.659, E3 +20783.248}
SPL {X  -159.317, Y  +686.157, Z    +0.000, E1   -18.660, E3 +20784.738}
SPL {X  -159.973, Y  +673.799, Z    +0.000, E1    -5.345, E3 +20785.187}
SPL {X  -159.990, Y  +669.500, Z    +0.000, E1    +0.000, E3 +20785.227}
SPL {X  -159.990, Y  +667.794, Z    +0.000, E1    +4.255, E3 +20785.238}
SPL {X  -159.990, Y  +664.091, Z    +0.000, E1   +14.928, E3 +20785.310}
SPL {X  -159.990, Y  +659.599, Z    +0.000, E1   +28.016, E3 +20785.480}
SPL {X  -159.990, Y  +652.711, Z    +0.000, E1   +44.293, E3 +20785.960}
SPL {X  -159.990, Y  +640.730, Z    +0.000, E1   +60.297, E3 +20787.309}
SPL {X  -159.990, Y  +620.478, Z    +0.000, E1   +70.026, E3 +20791.122}
SPL {X  -159.990, Y  +573.021, Z    +0.000, E1   +74.619, E3 +20805.066}
SPL {X  -154.165, Y  +339.724, Z    +0.000, E1   +75.927, E3 +20900.913}
SPL {X  -150.223, Y  +327.456, Z    +0.000, E1   +75.573, E3 +20911.178}
SPL {X  -136.549, Y  +299.126, Z    +0.000, E1   +77.537, E3 +20904.068}
ENDSPLINE

SPLINE
SPL {X  -136.862, Y  +299.641, Z    +0.000, E1   +76.604, E3 +20912.710}
ENDSPLINE

SPLINE
SPL {X  -136.434, Y  +298.938, Z    +0.000, E1   +75.982, E3 +20918.601}
SPL {X  -135.890, Y  +298.057, Z    +0.000, E1   +75.040, E3 +20927.067}
SPL {X  -134.349, Y  +295.626, Z    +0.000, E1   +74.322, E3 +20933.914}
SPL {X  -131.287, Y  +291.064, Z    +0.000, E1   +73.972, E3 +20938.727}
SPL {X  -128.265, Y  +286.871, Z    +0.000, E1   +73.613, E3 +20943.183}
SPL {X  -125.161, Y  +282.843, Z    +0.000, E1   +73.232, E3 +20947.454}
SPL {X  -122.038, Y  +279.042, Z    +0.000, E1   +72.832, E3 +20951.434}
SPL {X  -118.642, Y  +275.165, Z    +0.000, E1   +72.381, E3 +20955.398}
SPL {X   -66.040, Y  +236.776, Z    +0.000, E1   +55.694, E3 +21116.761}
ENDSPLINE

SPLINE
SPL {X  -127.452, Y  +285.790, Z    +0.000, E1   +56.591, E3 +21290.706}
SPL {X  -151.591, Y  +331.344, Z    +0.000, E1   +43.870, E3 +21306.806}
SPL {X  -158.135, Y  +358.205, Z    +0.000, E1   +26.984, E3 +21310.533}
SPL {X  -159.602, Y  +371.361, Z    +0.000, E1   +14.835, E3 +21311.429}
SPL {X  -159.981, Y  +380.818, Z    +0.000, E1    +4.512, E3 +21311.707}
SPL {X  -159.990, Y  +384.681, Z    +0.000, E1    -0.222, E3 +21311.736}
SPL {X  -159.990, Y  +387.626, Z    +0.000, E1    -8.190, E3 +21311.764}
SPL {X  -159.990, Y  +390.340, Z    +0.000, E1   -15.987, E3 +21311.829}
SPL {X  -159.990, Y  +394.216, Z    +0.000, E1   -27.062, E3 +21311.991}
SPL {X  -159.990, Y  +399.855, Z    +0.000, E1   -40.916, E3 +21312.362}
SPL {X  -159.990, Y  +405.475, Z    +0.000, E1   -51.039, E3 +21312.879}
SPL {X  -159.990, Y  +414.231, Z    +0.000, E1   -60.575, E3 +21314.063}
SPL {X  -159.990, Y  +462.953, Z    +0.000, E1   -73.611, E3 +21325.802}
SPL {X  -153.839, Y  +715.436, Z    +0.000, E1   -75.884, E3 +21428.233}
SPL {X  -149.923, Y  +727.355, Z    +0.000, E1   -75.515, E3 +21438.343}
SPL {X  -145.995, Y  +736.939, Z    +0.000, E1   -75.150, E3 +21447.077}
SPL {X  -141.012, Y  +747.080, Z    +0.000, E1   -74.661, E3 +21456.929}
SPL {X  -136.371, Y  +755.165, Z    +0.000, E1   -74.152, E3 +21465.215}
SPL {X  -133.102, Y  +760.274, Z    +0.000, E1   -73.777, E3 +21470.600}
SPL {X  -128.975, Y  +766.169, Z    +0.000, E1   -73.313, E3 +21476.875}
SPL {X  -124.947, Y  +771.425, Z    +0.000, E1   -72.782, E3 +21482.568}
SPL {X  -121.698, Y  +775.357, Z    +0.000, E1   -72.353, E3 +21486.763}
SPL {X  -118.622, Y  +778.858, Z    +0.000, E1   -71.924, E3 +21490.389}
SPL {X   -66.171, Y  +817.165, Z    +0.000, E1   -56.016, E3 +21641.747}
ENDSPLINE

SPLINE
SPL {X  -126.418, Y  +769.557, Z    +0.000, E1   -57.118, E3 +21824.989}
SPL {X  -148.476, Y  +731.097, Z    +0.000, E1   -47.824, E3 +21840.145}
SPL {X  -156.642, Y  +704.059, Z    +0.000, E1   -33.659, E3 +21844.786}
SPL {X  -159.317, Y  +686.157, Z    +0.000, E1   -18.660, E3 +21846.276}
SPL {X  -159.907, Y  +676.666, Z    +0.000, E1    -8.555, E3 +21846.674}
SPL {X  -159.990, Y  +669.586, Z    +0.000, E1    -0.216, E3 +21846.765}
SPL {X  -159.990, Y  +667.794, Z    +0.000, E1    +4.255, E3 +21846.776}
SPL {X  -159.990, Y  +664.091, Z    +0.000, E1   +14.928, E3 +21846.848}
SPL {X  -159.990, Y  +659.599, Z    +0.000, E1   +28.016, E3 +21847.019}
SPL {X  -159.990, Y  +652.711, Z    +0.000, E1   +44.293, E3 +21847.498}
SPL {X  -159.990, Y  +640.730, Z    +0.000, E1   +60.297, E3 +21848.847}
SPL {X  -159.990, Y  +620.478, Z    +0.000, E1   +70.026, E3 +21852.661}
SPL {X  -159.990, Y  +573.021, Z    +0.000, E1   +74.619, E3 +21866.604}
SPL {X  -154.165, Y  +339.724, Z    +0.000, E1   +75.927, E3 +21962.451}
SPL {X  -150.223, Y  +327.456, Z    +0.000, E1   +75.573, E3 +21972.716}
SPL {X  -136.549, Y  +299.126, Z    +0.000, E1   +77.537, E3 +21965.606}
ENDSPLINE

SPLINE
SPL {X  -136.862, Y  +299.641, Z    +0.000, E1   +76.604, E3 +21974.248}
ENDSPLINE

SPLINE
SPL {X  -136.434, Y  +298.938, Z    +0.000, E1   +75.982, E3 +21980.139}
SPL {X  -135.890, Y  +298.057, Z    +0.000, E1   +75.040, E3 +21988.605}
SPL {X  -134.349, Y  +295.626, Z    +0.000, E1   +74.322, E3 +21995.453}
SPL {X  -131.287, Y  +291.064, Z    +0.000, E1   +73.972, E3 +22000.265}
SPL {X  -128.265, Y  +286.871, Z    +0.000, E1   +73.613, E3 +22004.721}
SPL {X  -125.161, Y  +282.843, Z    +0.000, E1   +73.232, E3 +22008.993}
SPL {X  -122.038, Y  +279.042, Z    +0.000, E1   +72.832, E3 +22012.973}
SPL {X  -118.642, Y  +275.165, Z    +0.000, E1   +72.381, E3 +22016.936}
SPL {X   -66.040, Y  +236.776, Z    +0.000, E1   +55.694, E3 +22178.299}
ENDSPLINE

SPLINE
SPL {X  -127.452, Y  +285.790, Z    +0.000, E1   +56.591, E3 +22352.245}
SPL {X  -148.001, Y  +321.733, Z    +0.000, E1   +47.810, E3 +22366.348}
SPL {X  -154.604, Y  +341.337, Z    +0.000, E1   +38.630, E3 +22370.122}
SPL {X  -158.135, Y  +358.205, Z    +0.000, E1   +26.984, E3 +22372.072}
SPL {X  -159.602, Y  +371.361, Z    +0.000, E1   +14.835, E3 +22372.968}
SPL {X  -159.981, Y  +380.818, Z    +0.000, E1    +4.512, E3 +22373.246}
SPL {X  -159.990, Y  +384.681, Z    +0.000, E1    -0.222, E3 +22373.274}
SPL {X  -159.990, Y  +389.079, Z    +0.000, E1   -12.017, E3 +22373.337}
SPL {X  -159.990, Y  +394.216, Z    +0.000, E1   -27.062, E3 +22373.529}
SPL {X  -159.990, Y  +399.855, Z    +0.000, E1   -40.916, E3 +22373.900}
SPL {X  -159.990, Y  +405.475, Z    +0.000, E1   -51.039, E3 +22374.417}
SPL {X  -159.990, Y  +414.231, Z    +0.000, E1   -60.575, E3 +22375.602}
SPL {X  -159.990, Y  +462.953, Z    +0.000, E1   -73.611, E3 +22387.341}
SPL {X  -153.839, Y  +715.436, Z    +0.000, E1   -75.884, E3 +22489.771}
SPL {X  -148.840, Y  +730.182, Z    +0.000, E1   -75.434, E3 +22502.348}
SPL {X  -143.409, Y  +742.426, Z    +0.000, E1   -74.905, E3 +22513.860}
SPL {X  -139.557, Y  +749.735, Z    +0.000, E1   -74.483, E3 +22521.208}
SPL {X  -136.371, Y  +755.165, Z    +0.000, E1   -74.152, E3 +22526.753}
SPL {X  -133.102, Y  +760.274, Z    +0.000, E1   -73.777, E3 +22532.139}
SPL {X  -128.975, Y  +766.169, Z    +0.000, E1   -73.313, E3 +22538.414}
SPL {X  -124.947, Y  +771.425, Z    +0.000, E1   -72.782, E3 +22544.107}
SPL {X  -121.698, Y  +775.357, Z    +0.000, E1   -72.353, E3 +22548.301}
SPL {X  -118.622, Y  +778.858, Z    +0.000, E1   -71.924, E3 +22551.927}
SPL {X   -66.171, Y  +817.165, Z    +0.000, E1   -56.016, E3 +22703.286}
ENDSPLINE

SPLINE
SPL {X  -126.418, Y  +769.557, Z    +0.000, E1   -57.118, E3 +22886.527}
SPL {X  -145.244, Y  +738.589, Z    +0.000, E1   -50.405, E3 +22899.769}
SPL {X  -150.151, Y  +726.741, Z    +0.000, E1   -46.068, E3 +22902.695}
SPL {X  -156.642, Y  +704.059, Z    +0.000, E1   -33.659, E3 +22906.325}
SPL {X  -159.317, Y  +686.157, Z    +0.000, E1   -18.660, E3 +22907.815}
SPL {X  -159.973, Y  +673.799, Z    +0.000, E1    -5.345, E3 +22908.264}
SPL {X  -159.990, Y  +669.500, Z    +0.000, E1    +0.000, E3 +22908.304}
SPL {X  -159.990, Y  +667.794, Z    +0.000, E1    +4.255, E3 +22908.315}
SPL {X  -159.990, Y  +664.091, Z    +0.000, E1   +14.928, E3 +22908.387}
SPL {X  -159.990, Y  +658.301, Z    +0.000, E1   +31.283, E3 +22908.639}
SPL {X  -159.990, Y  +650.845, Z    +0.000, E1   +47.892, E3 +22909.185}
SPL {X  -159.990, Y  +640.730, Z    +0.000, E1   +60.297, E3 +22910.386}
SPL {X  -159.990, Y  +620.478, Z    +0.000, E1   +70.026, E3 +22914.199}
SPL {X  -159.990, Y  +573.021, Z    +0.000, E1   +74.619, E3 +22928.143}
SPL {X  -154.165, Y  +339.724, Z    +0.000, E1   +75.927, E3 +23023.990}
SPL {X  -150.223, Y  +327.456, Z    +0.000, E1   +75.573, E3 +23034.255}
SPL {X  -136.549, Y  +299.126, Z    +0.000, E1   +77.537, E3 +23027.145}
ENDSPLINE

SPLINE
SPL {X  -136.862, Y  +299.641, Z    +0.000, E1   +76.604, E3 +23035.787}
ENDSPLINE

SPLINE
SPL {X  -136.434, Y  +298.938, Z    +0.000, E1   +75.982, E3 +23041.678}
SPL {X  -135.890, Y  +298.057, Z    +0.000, E1   +75.040, E3 +23050.144}
SPL {X  -134.349, Y  +295.626, Z    +0.000, E1   +74.322, E3 +23056.991}
SPL {X  -131.287, Y  +291.064, Z    +0.000, E1   +73.972, E3 +23061.804}
SPL {X  -128.265, Y  +286.871, Z    +0.000, E1   +73.613, E3 +23066.260}
SPL {X  -125.161, Y  +282.843, Z    +0.000, E1   +73.232, E3 +23070.531}
SPL {X  -122.038, Y  +279.042, Z    +0.000, E1   +72.832, E3 +23074.511}
SPL {X  -118.642, Y  +275.165, Z    +0.000, E1   +72.381, E3 +23078.474}
SPL {X   -66.040, Y  +236.776, Z    +0.000, E1   +55.694, E3 +23239.838}
ENDSPLINE

SPLINE
SPL {X  -127.452, Y  +285.790, Z    +0.000, E1   +56.591, E3 +23413.783}
SPL {X  -148.001, Y  +321.733, Z    +0.000, E1   +47.810, E3 +23427.887}
SPL {X  -154.604, Y  +341.337, Z    +0.000, E1   +38.630, E3 +23431.660}
SPL {X  -158.135, Y  +358.205, Z    +0.000, E1   +26.984, E3 +23433.610}
SPL {X  -159.602, Y  +371.361, Z    +0.000, E1   +14.835, E3 +23434.506}
SPL {X  -159.981, Y  +380.818, Z    +0.000, E1    +4.512, E3 +23434.784}
SPL {X  -159.990, Y  +384.681, Z    +0.000, E1    -0.222, E3 +23434.813}
SPL {X  -159.990, Y  +389.079, Z    +0.000, E1   -12.017, E3 +23434.876}
SPL {X  -159.990, Y  +394.216, Z    +0.000, E1   -27.062, E3 +23435.068}
SPL {X  -159.990, Y  +399.855, Z    +0.000, E1   -40.916, E3 +23435.439}
SPL {X  -159.990, Y  +405.475, Z    +0.000, E1   -51.039, E3 +23435.956}
SPL {X  -159.990, Y  +414.231, Z    +0.000, E1   -60.575, E3 +23437.140}
SPL {X  -159.990, Y  +462.953, Z    +0.000, E1   -73.611, E3 +23448.879}
SPL {X  -153.839, Y  +715.436, Z    +0.000, E1   -75.884, E3 +23551.310}
SPL {X  -148.840, Y  +730.182, Z    +0.000, E1   -75.434, E3 +23563.886}
SPL {X  -143.409, Y  +742.426, Z    +0.000, E1   -74.905, E3 +23575.398}
SPL {X  -139.557, Y  +749.735, Z    +0.000, E1   -74.483, E3 +23582.746}
SPL {X  -136.371, Y  +755.165, Z    +0.000, E1   -74.152, E3 +23588.292}
SPL {X  -133.102, Y  +760.274, Z    +0.000, E1   -73.777, E3 +23593.677}
SPL {X  -128.975, Y  +766.169, Z    +0.000, E1   -73.313, E3 +23599.952}
SPL {X  -124.947, Y  +771.425, Z    +0.000, E1   -72.782, E3 +23605.645}
SPL {X  -121.698, Y  +775.357, Z    +0.000, E1   -72.353, E3 +23609.840}
SPL {X  -118.622, Y  +778.858, Z    +0.000, E1   -71.924, E3 +23613.466}
SPL {X   -66.171, Y  +817.165, Z    +0.000, E1   -56.016, E3 +23764.824}
ENDSPLINE

SPLINE
SPL {X  -126.418, Y  +769.557, Z    +0.000, E1   -57.118, E3 +23948.065}
SPL {X  -145.244, Y  +738.589, Z    +0.000, E1   -50.405, E3 +23961.307}
SPL {X  -150.151, Y  +726.741, Z    +0.000, E1   -46.068, E3 +23964.234}
SPL {X  -156.642, Y  +704.059, Z    +0.000, E1   -33.659, E3 +23967.863}
SPL {X  -159.317, Y  +686.157, Z    +0.000, E1   -18.660, E3 +23969.353}
SPL {X  -159.973, Y  +673.799, Z    +0.000, E1    -5.345, E3 +23969.802}
SPL {X  -159.990, Y  +669.500, Z    +0.000, E1    +0.000, E3 +23969.842}
SPL {X  -159.990, Y  +667.794, Z    +0.000, E1    +4.255, E3 +23969.853}
SPL {X  -159.990, Y  +664.091, Z    +0.000, E1   +14.928, E3 +23969.925}
SPL {X  -159.990, Y  +658.301, Z    +0.000, E1   +31.283, E3 +23970.178}
SPL {X  -159.990, Y  +650.845, Z    +0.000, E1   +47.892, E3 +23970.723}
SPL {X  -159.990, Y  +640.730, Z    +0.000, E1   +60.297, E3 +23971.924}
SPL {X  -159.990, Y  +620.478, Z    +0.000, E1   +70.026, E3 +23975.738}
SPL {X  -159.990, Y  +573.021, Z    +0.000, E1   +74.619, E3 +23989.681}
SPL {X  -154.165, Y  +339.724, Z    +0.000, E1   +75.927, E3 +24085.528}
SPL {X  -150.223, Y  +327.456, Z    +0.000, E1   +75.573, E3 +24095.793}
SPL {X  -136.549, Y  +299.126, Z    +0.000, E1   +77.537, E3 +24088.683}
ENDSPLINE

SPLINE
SPL {X  -136.862, Y  +299.641, Z    +0.000, E1   +76.604, E3 +24097.325}
ENDSPLINE

SPLINE
SPL {X  -136.434, Y  +298.938, Z    +0.000, E1   +75.982, E3 +24103.216}
SPL {X  -135.890, Y  +298.057, Z    +0.000, E1   +75.040, E3 +24111.682}
SPL {X  -134.349, Y  +295.626, Z    +0.000, E1   +74.322, E3 +24118.530}
SPL {X  -131.287, Y  +291.064, Z    +0.000, E1   +73.972, E3 +24123.342}
SPL {X  -128.265, Y  +286.871, Z    +0.000, E1   +73.613, E3 +24127.798}
SPL {X  -125.161, Y  +282.843, Z    +0.000, E1   +73.232, E3 +24132.070}
SPL {X  -122.038, Y  +279.042, Z    +0.000, E1   +72.832, E3 +24136.050}
SPL {X  -118.642, Y  +275.165, Z    +0.000, E1   +72.381, E3 +24140.013}
SPL {X   -66.040, Y  +236.776, Z    +0.000, E1   +55.694, E3 +24301.376}
ENDSPLINE

SPLINE
SPL {X  -127.452, Y  +285.790, Z    +0.000, E1   +56.591, E3 +24475.322}
SPL {X  -148.001, Y  +321.733, Z    +0.000, E1   +47.810, E3 +24489.425}
SPL {X  -154.604, Y  +341.337, Z    +0.000, E1   +38.630, E3 +24493.199}
SPL {X  -158.135, Y  +358.205, Z    +0.000, E1   +26.984, E3 +24495.149}
SPL {X  -159.602, Y  +371.361, Z    +0.000, E1   +14.835, E3 +24496.045}
SPL {X  -159.981, Y  +380.818, Z    +0.000, E1    +4.512, E3 +24496.322}
SPL {X  -159.990, Y  +384.681, Z    +0.000, E1    -0.222, E3 +24496.351}
SPL {X  -159.990, Y  +389.079, Z    +0.000, E1   -12.017, E3 +24496.414}
SPL {X  -159.990, Y  +394.216, Z    +0.000, E1   -27.062, E3 +24496.606}
SPL {X  -159.990, Y  +399.855, Z    +0.000, E1   -40.916, E3 +24496.977}
SPL {X  -159.990, Y  +405.475, Z    +0.000, E1   -51.039, E3 +24497.494}
SPL {X  -159.990, Y  +414.231, Z    +0.000, E1   -60.575, E3 +24498.678}
SPL {X  -159.990, Y  +462.953, Z    +0.000, E1   -73.611, E3 +24510.417}
SPL {X  -153.839, Y  +715.436, Z    +0.000, E1   -75.884, E3 +24612.848}
SPL {X  -148.840, Y  +730.182, Z    +0.000, E1   -75.434, E3 +24625.425}
SPL {X  -143.409, Y  +742.426, Z    +0.000, E1   -74.905, E3 +24636.937}
SPL {X  -139.557, Y  +749.735, Z    +0.000, E1   -74.483, E3 +24644.285}
SPL {X  -136.371, Y  +755.165, Z    +0.000, E1   -74.152, E3 +24649.830}
SPL {X  -133.102, Y  +760.274, Z    +0.000, E1   -73.777, E3 +24655.215}
SPL {X  -128.975, Y  +766.169, Z    +0.000, E1   -73.313, E3 +24661.491}
SPL {X  -124.947, Y  +771.425, Z    +0.000, E1   -72.782, E3 +24667.184}
SPL {X  -121.698, Y  +775.357, Z    +0.000, E1   -72.353, E3 +24671.378}
SPL {X  -118.622, Y  +778.858, Z    +0.000, E1   -71.924, E3 +24675.004}
SPL {X   -66.171, Y  +817.165, Z    +0.000, E1   -56.016, E3 +24826.363}
ENDSPLINE

SPLINE
SPL {X  -126.418, Y  +769.557, Z    +0.000, E1   -57.118, E3 +25009.604}
SPL {X  -145.244, Y  +738.589, Z    +0.000, E1   -50.405, E3 +25022.845}
SPL {X  -150.151, Y  +726.741, Z    +0.000, E1   -46.068, E3 +25025.772}
SPL {X  -156.642, Y  +704.059, Z    +0.000, E1   -33.659, E3 +25029.402}
SPL {X  -159.317, Y  +686.157, Z    +0.000, E1   -18.660, E3 +25030.892}
SPL {X  -159.973, Y  +673.799, Z    +0.000, E1    -5.345, E3 +25031.340}
SPL {X  -159.990, Y  +669.500, Z    +0.000, E1    +0.000, E3 +25031.381}
SPL {X  -159.990, Y  +667.794, Z    +0.000, E1    +4.255, E3 +25031.392}
SPL {X  -159.990, Y  +664.091, Z    +0.000, E1   +14.928, E3 +25031.464}
SPL {X  -159.990, Y  +658.301, Z    +0.000, E1   +31.283, E3 +25031.716}
SPL {X  -159.990, Y  +650.845, Z    +0.000, E1   +47.892, E3 +25032.262}
SPL {X  -159.990, Y  +640.730, Z    +0.000, E1   +60.297, E3 +25033.463}
SPL {X  -159.990, Y  +620.478, Z    +0.000, E1   +70.026, E3 +25037.276}
SPL {X  -159.990, Y  +573.021, Z    +0.000, E1   +74.619, E3 +25051.220}
SPL {X  -154.165, Y  +339.724, Z    +0.000, E1   +75.927, E3 +25147.067}
SPL {X  -150.223, Y  +327.456, Z    +0.000, E1   +75.573, E3 +25157.332}
SPL {X  -136.549, Y  +299.126, Z    +0.000, E1   +77.537, E3 +25150.222}
ENDSPLINE

SPLINE
SPL {X  -136.626, Y  +299.252, Z    +0.000, E1   +76.314, E3 +25161.872}
ENDSPLINE

SPLINE
SPL {X  -135.890, Y  +298.057, Z    +0.000, E1   +75.040, E3 +25173.221}
SPL {X  -134.349, Y  +295.626, Z    +0.000, E1   +74.322, E3 +25180.068}
SPL {X  -131.287, Y  +291.064, Z    +0.000, E1   +73.972, E3 +25184.881}
SPL {X  -128.265, Y  +286.871, Z    +0.000, E1   +73.613, E3 +25189.337}
SPL {X  -125.161, Y  +282.843, Z    +0.000, E1   +73.232, E3 +25193.608}
SPL {X  -122.038, Y  +279.042, Z    +0.000, E1   +72.832, E3 +25197.588}
SPL {X  -118.642, Y  +275.165, Z    +0.000, E1   +72.381, E3 +25201.551}
SPL {X   -66.040, Y  +236.776, Z    +0.000, E1   +55.694, E3 +25362.915}
ENDSPLINE

SPLINE
SPL {X  -127.452, Y  +285.790, Z    +0.000, E1   +56.591, E3 +25536.860}
SPL {X  -151.591, Y  +331.344, Z    +0.000, E1   +43.870, E3 +25552.959}
SPL {X  -158.135, Y  +358.205, Z    +0.000, E1   +26.984, E3 +25556.687}
SPL {X  -159.602, Y  +371.361, Z    +0.000, E1   +14.835, E3 +25557.583}
SPL {X  -159.981, Y  +380.818, Z    +0.000, E1    +4.512, E3 +25557.861}
SPL {X  -159.990, Y  +384.681, Z    +0.000, E1    -0.222, E3 +25557.890}
SPL {X  -159.990, Y  +387.626, Z    +0.000, E1    -8.190, E3 +25557.918}
SPL {X  -159.990, Y  +390.340, Z    +0.000, E1   -15.987, E3 +25557.983}
SPL {X  -159.990, Y  +394.216, Z    +0.000, E1   -27.062, E3 +25558.145}
SPL {X  -159.990, Y  +399.855, Z    +0.000, E1   -40.916, E3 +25558.516}
SPL {X  -159.990, Y  +405.475, Z    +0.000, E1   -51.039, E3 +25559.033}
SPL {X  -159.990, Y  +414.231, Z    +0.000, E1   -60.575, E3 +25560.217}
SPL {X  -159.990, Y  +462.953, Z    +0.000, E1   -73.611, E3 +25571.956}
SPL {X  -153.839, Y  +715.436, Z    +0.000, E1   -75.884, E3 +25674.386}
SPL {X  -149.923, Y  +727.355, Z    +0.000, E1   -75.515, E3 +25684.496}
SPL {X  -145.995, Y  +736.939, Z    +0.000, E1   -75.150, E3 +25693.231}
SPL {X  -142.305, Y  +744.618, Z    +0.000, E1   -74.773, E3 +25700.675}
SPL {X  -139.557, Y  +749.735, Z    +0.000, E1   -74.483, E3 +25705.823}
SPL {X  -136.371, Y  +755.165, Z    +0.000, E1   -74.152, E3 +25711.369}
SPL {X  -131.455, Y  +762.694, Z    +0.000, E1   -73.615, E3 +25719.287}
SPL {X  -125.933, Y  +770.180, Z    +0.000, E1   -72.934, E3 +25727.352}
SPL {X  -121.698, Y  +775.357, Z    +0.000, E1   -72.353, E3 +25732.917}
SPL {X  -118.622, Y  +778.858, Z    +0.000, E1   -71.924, E3 +25736.543}
SPL {X   -66.171, Y  +817.165, Z    +0.000, E1   -56.016, E3 +25887.901}
ENDSPLINE

SPLINE
SPL {X  -126.418, Y  +769.557, Z    +0.000, E1   -57.118, E3 +26071.142}
SPL {X  -145.244, Y  +738.589, Z    +0.000, E1   -50.405, E3 +26084.384}
SPL {X  -150.151, Y  +726.741, Z    +0.000, E1   -46.068, E3 +26087.311}
SPL {X  -156.642, Y  +704.059, Z    +0.000, E1   -33.659, E3 +26090.940}
SPL {X  -159.317, Y  +686.157, Z    +0.000, E1   -18.660, E3 +26092.430}
SPL {X  -159.973, Y  +673.799, Z    +0.000, E1    -5.345, E3 +26092.879}
SPL {X  -159.990, Y  +669.500, Z    +0.000, E1    +0.000, E3 +26092.919}
SPL {X  -159.990, Y  +667.794, Z    +0.000, E1    +4.255, E3 +26092.930}
SPL {X  -159.990, Y  +664.091, Z    +0.000, E1   +14.928, E3 +26093.002}
SPL {X  -159.990, Y  +659.599, Z    +0.000, E1   +28.016, E3 +26093.173}
SPL {X  -159.990, Y  +652.711, Z    +0.000, E1   +44.293, E3 +26093.652}
SPL {X  -159.990, Y  +640.730, Z    +0.000, E1   +60.297, E3 +26095.001}
SPL {X  -159.990, Y  +620.478, Z    +0.000, E1   +70.026, E3 +26098.814}
SPL {X  -159.990, Y  +573.021, Z    +0.000, E1   +74.619, E3 +26112.758}
SPL {X  -154.165, Y  +339.724, Z    +0.000, E1   +75.927, E3 +26208.605}
SPL {X  -150.571, Y  +328.416, Z    +0.000, E1   +75.599, E3 +26218.051}
SPL {X  -148.206, Y  +322.236, Z    +0.000, E1   +75.365, E3 +26223.595}
SPL {X  -136.549, Y  +299.126, Z    +0.000, E1   +77.537, E3 +26211.760}
ENDSPLINE

SPLINE
SPL {X  -136.862, Y  +299.641, Z    +0.000, E1   +76.604, E3 +26220.402}
ENDSPLINE

SPLINE
SPL {X  -136.434, Y  +298.938, Z    +0.000, E1   +75.982, E3 +26226.293}
SPL {X  -135.890, Y  +298.057, Z    +0.000, E1   +75.040, E3 +26234.759}
SPL {X  -134.349, Y  +295.626, Z    +0.000, E1   +74.322, E3 +26241.606}
SPL {X  -131.287, Y  +291.064, Z    +0.000, E1   +73.972, E3 +26246.419}
SPL {X  -128.265, Y  +286.871, Z    +0.000, E1   +73.613, E3 +26250.875}
SPL {X  -125.161, Y  +282.843, Z    +0.000, E1   +73.232, E3 +26255.147}
SPL {X  -122.038, Y  +279.042, Z    +0.000, E1   +72.832, E3 +26259.127}
SPL {X  -118.642, Y  +275.165, Z    +0.000, E1   +72.381, E3 +26263.090}
SPL {X   -66.040, Y  +236.776, Z    +0.000, E1   +55.694, E3 +26424.453}
ENDSPLINE

SPLINE
SPL {X  -127.452, Y  +285.790, Z    +0.000, E1   +56.591, E3 +26598.399}
SPL {X  -151.591, Y  +331.344, Z    +0.000, E1   +43.870, E3 +26614.498}
SPL {X  -158.135, Y  +358.205, Z    +0.000, E1   +26.984, E3 +26618.226}
SPL {X  -159.602, Y  +371.361, Z    +0.000, E1   +14.835, E3 +26619.122}
SPL {X  -159.981, Y  +380.818, Z    +0.000, E1    +4.512, E3 +26619.399}
SPL {X  -159.990, Y  +384.681, Z    +0.000, E1    -0.222, E3 +26619.428}
SPL {X  -159.990, Y  +389.079, Z    +0.000, E1   -12.017, E3 +26619.491}
SPL {X  -159.990, Y  +394.216, Z    +0.000, E1   -27.062, E3 +26619.683}
SPL {X  -159.990, Y  +399.855, Z    +0.000, E1   -40.916, E3 +26620.054}
SPL {X  -159.990, Y  +405.475, Z    +0.000, E1   -51.039, E3 +26620.571}
SPL {X  -159.990, Y  +414.231, Z    +0.000, E1   -60.575, E3 +26621.755}
SPL {X  -159.990, Y  +462.953, Z    +0.000, E1   -73.611, E3 +26633.494}
SPL {X  -153.839, Y  +715.436, Z    +0.000, E1   -75.884, E3 +26735.925}
SPL {X  -148.840, Y  +730.182, Z    +0.000, E1   -75.434, E3 +26748.502}
SPL {X  -143.409, Y  +742.426, Z    +0.000, E1   -74.905, E3 +26760.014}
SPL {X  -139.557, Y  +749.735, Z    +0.000, E1   -74.483, E3 +26767.362}
SPL {X  -136.371, Y  +755.165, Z    +0.000, E1   -74.152, E3 +26772.907}
SPL {X  -133.102, Y  +760.274, Z    +0.000, E1   -73.777, E3 +26778.292}
SPL {X  -128.975, Y  +766.169, Z    +0.000, E1   -73.313, E3 +26784.568}
SPL {X  -124.947, Y  +771.425, Z    +0.000, E1   -72.782, E3 +26790.261}
SPL {X  -121.698, Y  +775.357, Z    +0.000, E1   -72.353, E3 +26794.455}
SPL {X  -118.622, Y  +778.858, Z    +0.000, E1   -71.924, E3 +26798.081}
SPL {X   -66.171, Y  +817.165, Z    +0.000, E1   -56.016, E3 +26949.440}
ENDSPLINE

SPLINE
SPL {X  -126.418, Y  +769.557, Z    +0.000, E1   -57.118, E3 +27132.681}
SPL {X  -145.244, Y  +738.589, Z    +0.000, E1   -50.405, E3 +27145.922}
SPL {X  -150.151, Y  +726.741, Z    +0.000, E1   -46.068, E3 +27148.849}
SPL {X  -156.642, Y  +704.059, Z    +0.000, E1   -33.659, E3 +27152.479}
SPL {X  -159.317, Y  +686.157, Z    +0.000, E1   -18.660, E3 +27153.969}
SPL {X  -159.973, Y  +673.799, Z    +0.000, E1    -5.345, E3 +27154.417}
SPL {X  -159.990, Y  +669.500, Z    +0.000, E1    +0.000, E3 +27154.457}
SPL {X  -159.990, Y  +667.794, Z    +0.000, E1    +4.255, E3 +27154.469}
SPL {X  -159.990, Y  +664.091, Z    +0.000, E1   +14.928, E3 +27154.541}
SPL {X  -159.990, Y  +658.301, Z    +0.000, E1   +31.283, E3 +27154.793}
SPL {X  -159.990, Y  +650.845, Z    +0.000, E1   +47.892, E3 +27155.338}
SPL {X  -159.990, Y  +640.730, Z    +0.000, E1   +60.297, E3 +27156.540}
SPL {X  -159.990, Y  +620.478, Z    +0.000, E1   +70.026, E3 +27160.353}
SPL {X  -159.990, Y  +573.021, Z    +0.000, E1   +74.619, E3 +27174.297}
SPL {X  -154.165, Y  +339.724, Z    +0.000, E1   +75.927, E3 +27270.144}
SPL {X  -150.223, Y  +327.456, Z    +0.000, E1   +75.573, E3 +27280.409}
SPL {X  -136.549, Y  +299.126, Z    +0.000, E1   +77.537, E3 +27273.299}
ENDSPLINE

SPLINE
SPL {X  -136.862, Y  +299.641, Z    +0.000, E1   +76.604, E3 +27281.941}
ENDSPLINE

SPLINE
SPL {X  -136.434, Y  +298.938, Z    +0.000, E1   +75.982, E3 +27287.832}
SPL {X  -135.890, Y  +298.057, Z    +0.000, E1   +75.040, E3 +27296.298}
SPL {X  -134.349, Y  +295.626, Z    +0.000, E1   +74.322, E3 +27303.145}
SPL {X  -131.287, Y  +291.064, Z    +0.000, E1   +73.972, E3 +27307.957}
SPL {X  -128.265, Y  +286.871, Z    +0.000, E1   +73.613, E3 +27312.413}
SPL {X  -125.161, Y  +282.843, Z    +0.000, E1   +73.232, E3 +27316.685}
SPL {X  -122.038, Y  +279.042, Z    +0.000, E1   +72.832, E3 +27320.665}
SPL {X  -118.642, Y  +275.165, Z    +0.000, E1   +72.381, E3 +27324.628}
SPL {X   -66.040, Y  +236.776, Z    +0.000, E1   +55.694, E3 +27485.992}
ENDSPLINE

